LIN {X 0,Y 629.208,Z 740.926,A -85,B 0,C 180,E1 29271.292,E2 29271.292} C_VEL
LIN {X 0,Y 628.174,Z 758.568,A -85,B 0,C 180,E1 29269.915,E2 29269.915} C_VEL
LIN {X 0,Y 627.247,Z 774.118,A -85,B 0,C 180,E1 29268.495,E2 29268.495} C_VEL
LIN {X 0,Y 626.389,Z 788.139,A -85,B 0,C 180,E1 29266.985,E2 29266.985} C_VEL
LIN {X 0,Y 625.582,Z 802.216,A -85,B 0,C 180,E1 29265.196,E2 29265.196} C_VEL
LIN {X 0,Y 624.988,Z 813.341,A -85,B 0,C 180,E1 29263.508,E2 29263.508} C_VEL
LIN {X 0,Y 624.565,Z 822.244,A -85,B 0,C 180,E1 29261.919,E2 29261.919} C_VEL
LIN {X 0,Y 624.211,Z 832.3,A -85,B 0,C 180,E1 29259.776,E2 29259.776} C_VEL
LIN {X 0,Y 624.048,Z 838.961,A -85,B 0,C 180,E1 29258.013,E2 29258.013} C_VEL
LIN {X 0,Y 623.969,Z 843.988,A -85,B 0,C 180,E1 29256.348,E2 29256.348} C_VEL
LIN {X 0,Y 623.918,Z 847.629,A -85,B 0,C 180,E1 29254.78,E2 29254.78} C_VEL
LIN {X 0,Y 623.903,Z 850.253,A -85,B 0,C 180,E1 29253.193,E2 29253.193} C_VEL
LIN {X 0,Y 623.908,Z 851.807,A -85,B 0,C 180,E1 29251.653,E2 29251.653} C_VEL
LIN {X 0,Y 623.919,Z 852.393,A -85,B 0,C 180,E1 29250,E2 29250} C_VEL
LIN {X 0,Y 623.906,Z 851.865,A -85,B 0,C 180,E1 29248.347,E2 29248.347} C_VEL
LIN {X 0,Y 623.901,Z 850.34,A -85,B 0,C 180,E1 29246.785,E2 29246.785} C_VEL
LIN {X 0,Y 623.92,Z 847.804,A -85,B 0,C 180,E1 29245.22,E2 29245.22} C_VEL
LIN {X 0,Y 623.969,Z 844.223,A -85,B 0,C 180,E1 29243.652,E2 29243.652} C_VEL
LIN {X 0,Y 624.029,Z 839.56,A -85,B 0,C 180,E1 29242.08,E2 29242.08} C_VEL
LIN {X 0,Y 624.164,Z 833.767,A -85,B 0,C 180,E1 29240.503,E2 29240.503} C_VEL
LIN {X 0,Y 624.432,Z 825.538,A -85,B 0,C 180,E1 29238.641,E2 29238.641} C_VEL
LIN {X 0,Y 624.9,Z 815.025,A -85,B 0,C 180,E1 29236.679,E2 29236.679} C_VEL
LIN {X 0,Y 625.468,Z 804.166,A -85,B 0,C 180,E1 29234.991,E2 29234.991} C_VEL
LIN {X 0,Y 626.179,Z 791.739,A -85,B 0,C 180,E1 29233.354,E2 29233.354} C_VEL
LIN {X 0,Y 627.018,Z 777.74,A -85,B 0,C 180,E1 29231.787,E2 29231.787} C_VEL
LIN {X 0,Y 627.946,Z 762.367,A -85,B 0,C 180,E1 29230.32,E2 29230.32} C_VEL
LIN {X 0,Y 628.974,Z 745.456,A -85,B 0,C 180,E1 29228.944,E2 29228.944} C_VEL
LIN {X 0,Y 629.98,Z 727.417,A -85,B 0,C 180,E1 29227.708,E2 29227.708} C_VEL
LIN {X 0,Y 630.985,Z 708.54,A -85,B 0,C 180,E1 29226.612,E2 29226.612} C_VEL
LIN {X 0,Y 631.859,Z 689.995,A -85,B 0,C 180,E1 29225.705,E2 29225.705} C_VEL
LIN {X 0,Y 632.742,Z 669.051,A -85,B 0,C 180,E1 29224.87,E2 29224.87} C_VEL
LIN {X 0,Y 633.413,Z 648.623,A -85,B 0,C 180,E1 29224.226,E2 29224.226} C_VEL
LIN {X 0,Y 634.025,Z 626.542,A -85,B 0,C 180,E1 29223.692,E2 29223.692} C_VEL
LIN {X 0,Y 634.453,Z 605.1,A -85,B 0,C 180,E1 29223.321,E2 29223.321} C_VEL
LIN {X 0,Y 638.365,Z 407.202,A -85,B 0,C 180,E1 29220.608,E2 29220.608} C_VEL
LIN {X 0,Y 639.37,Z 326.363,A -85,B 0,C 180,E1 29219.579,E2 29219.579} C_VEL
LIN {X 0,Y 639.015,Z 324.152,A -85,B 0,C 180,E1 29219.511,E2 29219.511} C_VEL
LIN {X 0,Y 639.079,Z 296.354,A -85,B 0,C 180,E1 29217.65,E2 29217.65} C_VEL
LIN {X 0,Y 640.388,Z 256.622,A -85,B 0,C 180,E1 29214.747,E2 29214.747} C_VEL
LIN {X 0,Y 640.643,Z 246.721,A -85,B 0,C 180,E1 29214.024,E2 29214.024} C_VEL
LIN {X 0,Y 633.821,Z 228.869,A -85,B 0,C 180,E1 29212.219,E2 29212.219} C_VEL
LIN {X 0,Y 627.274,Z 213.434,A -85,B 0,C 180,E1 29210.706,E2 29210.706} C_VEL
LIN {X 0,Y 624.952,Z 207.388,A -85,B 0,C 180,E1 29210.129,E2 29210.129} C_VEL
LIN {X 0,Y 624.924,Z 207.385,A -85,B 0,C 180,E1 29206.988,E2 29206.988} C_VEL
LIN {X 0,Y 624.946,Z 207.377,A -85,B 0,C 180,E1 29203.851,E2 29203.851} C_VEL
LIN {X 0,Y 624.928,Z 207.382,A -85,B 0,C 180,E1 29200.754,E2 29200.754} C_VEL
LIN {X 0,Y 624.947,Z 207.376,A -85,B 0,C 180,E1 29197.629,E2 29197.629} C_VEL
LIN {X 0,Y 624.94,Z 207.389,A -85,B 0,C 180,E1 29194.499,E2 29194.499} C_VEL
LIN {X 0,Y 624.947,Z 207.379,A -85,B 0,C 180,E1 29191.224,E2 29191.224} C_VEL
LIN {X 0,Y 624.945,Z 207.373,A -85,B 0,C 180,E1 29188.06,E2 29188.06} C_VEL
LIN {X 0,Y 624.937,Z 207.381,A -85,B 0,C 180,E1 29184.88,E2 29184.88} C_VEL
LIN {X 0,Y 624.937,Z 207.383,A -85,B 0,C 180,E1 29181.79,E2 29181.79} C_VEL
LIN {X 0,Y 624.937,Z 207.371,A -85,B 0,C 180,E1 29178.663,E2 29178.663} C_VEL
LIN {X 0,Y 624.934,Z 207.381,A -85,B 0,C 180,E1 29175.593,E2 29175.593} C_VEL
LIN {X 0,Y 624.941,Z 207.366,A -85,B 0,C 180,E1 29172.474,E2 29172.474} C_VEL
LIN {X 0,Y 624.942,Z 207.38,A -85,B 0,C 180,E1 29169.3,E2 29169.3} C_VEL
LIN {X 0,Y 624.943,Z 207.365,A -85,B 0,C 180,E1 29166.062,E2 29166.062} C_VEL
LIN {X 0,Y 624.947,Z 207.38,A -85,B 0,C 180,E1 29162.843,E2 29162.843} C_VEL
LIN {X 0,Y 624.923,Z 207.363,A -85,B 0,C 180,E1 29159.725,E2 29159.725} C_VEL
LIN {X 0,Y 624.946,Z 207.381,A -85,B 0,C 180,E1 29156.606,E2 29156.606} C_VEL
LIN {X 0,Y 624.919,Z 207.364,A -85,B 0,C 180,E1 29153.477,E2 29153.477} C_VEL
LIN {X 0,Y 624.949,Z 207.381,A -85,B 0,C 180,E1 29150.329,E2 29150.329} C_VEL
LIN {X 0,Y 624.924,Z 207.382,A -85,B 0,C 180,E1 29147.244,E2 29147.244} C_VEL
LIN {X 0,Y 624.942,Z 207.385,A -85,B 0,C 180,E1 29144.026,E2 29144.026} C_VEL
LIN {X 0,Y 624.946,Z 207.377,A -85,B 0,C 180,E1 29140.853,E2 29140.853} C_VEL
LIN {X 0,Y 624.916,Z 207.388,A -85,B 0,C 180,E1 29137.642,E2 29137.642} C_VEL
LIN {X 0,Y 624.953,Z 207.381,A -85,B 0,C 180,E1 29134.609,E2 29134.609} C_VEL
LIN {X 0,Y 624.91,Z 207.385,A -85,B 0,C 180,E1 29131.454,E2 29131.454} C_VEL
LIN {X 0,Y 624.957,Z 207.381,A -85,B 0,C 180,E1 29128.454,E2 29128.454} C_VEL
LIN {X 0,Y 624.906,Z 207.388,A -85,B 0,C 180,E1 29125.329,E2 29125.329} C_VEL
LIN {X 0,Y 624.957,Z 207.38,A -85,B 0,C 180,E1 29122.209,E2 29122.209} C_VEL
LIN {X 0,Y 624.903,Z 207.389,A -85,B 0,C 180,E1 29119.186,E2 29119.186} C_VEL
LIN {X 0,Y 624.95,Z 207.462,A -85,B 0,C 180,E1 29116.613,E2 29116.613} C_VEL
LIN {X 0,Y 626.289,Z 210.904,A -85,B 0,C 180,E1 29116.267,E2 29116.267} C_VEL
LIN {X 0,Y 627.344,Z 212.887,A -85,B 0,C 180,E1 29116.043,E2 29116.043} C_VEL
LIN {X 0,Y 638.156,Z 234.423,A -85,B 0,C 180,E1 29113.754,E2 29113.754} C_VEL
LIN {X 0,Y 647.363,Z 253.935,A -85,B 0,C 180,E1 29111.855,E2 29111.855} C_VEL
LIN {X 0,Y 644.416,Z 304.648,A -85,B 0,C 180,E1 29109.218,E2 29109.218} C_VEL
LIN {X 0,Y 646.898,Z 323.157,A -85,B 0,C 180,E1 29108.795,E2 29108.795} C_VEL
LIN {X 0,Y 644.169,Z 514.087,A -85,B 0,C 180,E1 29106.373,E2 29106.373} C_VEL
LIN {X 0,Y 641.865,Z 692.934,A -85,B 0,C 180,E1 29104.147,E2 29104.147} C_VEL
LIN {X 0,Y 641.079,Z 718.1,A -85,B 0,C 180,E1 29103.674,E2 29103.674} C_VEL
LIN {X 0,Y 640.186,Z 739.868,A -85,B 0,C 180,E1 29103.131,E2 29103.131} C_VEL
LIN {X 0,Y 638.916,Z 765.321,A -85,B 0,C 180,E1 29102.318,E2 29102.318} C_VEL
LIN {X 0,Y 637.689,Z 787.238,A -85,B 0,C 180,E1 29101.461,E2 29101.461} C_VEL
LIN {X 0,Y 636.241,Z 810.546,A -85,B 0,C 180,E1 29100.369,E2 29100.369} C_VEL
LIN {X 0,Y 634.874,Z 830.591,A -85,B 0,C 180,E1 29099.276,E2 29099.276} C_VEL
LIN {X 0,Y 633.292,Z 852.909,A -85,B 0,C 180,E1 29097.862,E2 29097.862} C_VEL
LIN {X 0,Y 632.055,Z 867.818,A -85,B 0,C 180,E1 29096.748,E2 29096.748} C_VEL
LIN {X 0,Y 630.517,Z 886.159,A -85,B 0,C 180,E1 29095.202,E2 29095.202} C_VEL
LIN {X 0,Y 629.035,Z 903.822,A -85,B 0,C 180,E1 29093.482,E2 29093.482} C_VEL
LIN {X 0,Y 627.829,Z 919.315,A -85,B 0,C 180,E1 29091.782,E2 29091.782} C_VEL
LIN {X 0,Y 626.714,Z 934.515,A -85,B 0,C 180,E1 29089.867,E2 29089.867} C_VEL
LIN {X 0,Y 625.867,Z 947.149,A -85,B 0,C 180,E1 29088.055,E2 29088.055} C_VEL
LIN {X 0,Y 625.118,Z 960.283,A -85,B 0,C 180,E1 29085.874,E2 29085.874} C_VEL
LIN {X 0,Y 624.657,Z 970.018,A -85,B 0,C 180,E1 29083.987,E2 29083.987} C_VEL
LIN {X 0,Y 624.293,Z 979.836,A -85,B 0,C 180,E1 29081.736,E2 29081.736} C_VEL
LIN {X 0,Y 624.094,Z 986.816,A -85,B 0,C 180,E1 29079.778,E2 29079.778} C_VEL
LIN {X 0,Y 623.952,Z 993.243,A -85,B 0,C 180,E1 29077.551,E2 29077.551} C_VEL
LIN {X 0,Y 623.905,Z 997.655,A -85,B 0,C 180,E1 29075.426,E2 29075.426} C_VEL
LIN {X 0,Y 623.91,Z 1000.464,A -85,B 0,C 180,E1 29073.491,E2 29073.491} C_VEL
LIN {X 0,Y 623.909,Z 1002.214,A -85,B 0,C 180,E1 29071.194,E2 29071.194} C_VEL
LIN {X 0,Y 623.885,Z 1002.327,A -85,B 0,C 180,E1 29069.265,E2 29069.265} C_VEL
LIN {X 0,Y 623.889,Z 1001.292,A -85,B 0,C 180,E1 29067.336,E2 29067.336} C_VEL
LIN {X 0,Y 623.901,Z 998.451,A -85,B 0,C 180,E1 29065.035,E2 29065.035} C_VEL
LIN {X 0,Y 623.959,Z 994.689,A -85,B 0,C 180,E1 29063.097,E2 29063.097} C_VEL
LIN {X 0,Y 624.042,Z 988.934,A -85,B 0,C 180,E1 29060.873,E2 29060.873} C_VEL
LIN {X 0,Y 624.217,Z 981.602,A -85,B 0,C 180,E1 29058.73,E2 29058.73} C_VEL
LIN {X 0,Y 624.519,Z 973.532,A -85,B 0,C 180,E1 29056.765,E2 29056.765} C_VEL
LIN {X 0,Y 624.996,Z 962.86,A -85,B 0,C 180,E1 29054.599,E2 29054.599} C_VEL
LIN {X 0,Y 625.602,Z 951.969,A -85,B 0,C 180,E1 29052.706,E2 29052.706} C_VEL
LIN {X 0,Y 626.517,Z 937.317,A -85,B 0,C 180,E1 29050.515,E2 29050.515} C_VEL
LIN {X 0,Y 627.462,Z 924.012,A -85,B 0,C 180,E1 29048.785,E2 29048.785} C_VEL
LIN {X 0,Y 628.838,Z 906.301,A -85,B 0,C 180,E1 29046.775,E2 29046.775} C_VEL
LIN {X 0,Y 630.114,Z 890.795,A -85,B 0,C 180,E1 29045.233,E2 29045.233} C_VEL
LIN {X 0,Y 631.805,Z 870.854,A -85,B 0,C 180,E1 29043.494,E2 29043.494} C_VEL
LIN {X 0,Y 633.107,Z 855.309,A -85,B 0,C 180,E1 29042.307,E2 29042.307} C_VEL
LIN {X 0,Y 634.055,Z 841.543,A -85,B 0,C 180,E1 29041.405,E2 29041.405} C_VEL
LIN {X 0,Y 635.449,Z 820.222,A -85,B 0,C 180,E1 29040.183,E2 29040.183} C_VEL
LIN {X 0,Y 636.697,Z 797.901,A -85,B 0,C 180,E1 29039.101,E2 29039.101} C_VEL
LIN {X 0,Y 637.906,Z 775.285,A -85,B 0,C 180,E1 29038.165,E2 29038.165} C_VEL
LIN {X 0,Y 638.944,Z 751.93,A -85,B 0,C 180,E1 29037.377,E2 29037.377} C_VEL
LIN {X 0,Y 639.847,Z 727.921,A -85,B 0,C 180,E1 29036.72,E2 29036.72} C_VEL
LIN {X 0,Y 640.534,Z 703.096,A -85,B 0,C 180,E1 29036.219,E2 29036.219} C_VEL
LIN {X 0,Y 640.998,Z 677.434,A -85,B 0,C 180,E1 29035.856,E2 29035.856} C_VEL
LIN {X 0,Y 642.199,Z 471.258,A -85,B 0,C 180,E1 29033.497,E2 29033.497} C_VEL
LIN {X 0,Y 643.617,Z 320.826,A -85,B 0,C 180,E1 29031.652,E2 29031.652} C_VEL
LIN {X 0,Y 642.214,Z 312.028,A -85,B 0,C 180,E1 29031.452,E2 29031.452} C_VEL
LIN {X 0,Y 644.812,Z 281.295,A -85,B 0,C 180,E1 29029.712,E2 29029.712} C_VEL
LIN {X 0,Y 648.358,Z 254.707,A -85,B 0,C 180,E1 29028.05,E2 29028.05} C_VEL
LIN {X 0,Y 645.178,Z 246.171,A -85,B 0,C 180,E1 29026.883,E2 29026.883} C_VEL
LIN {X 0,Y 642.634,Z 240.116,A -85,B 0,C 180,E1 29025.809,E2 29025.809} C_VEL
LIN {X 0,Y 641.16,Z 236.75,A -85,B 0,C 180,E1 29025.053,E2 29025.053} C_VEL
LIN {X 0,Y 639.826,Z 233.597,A -85,B 0,C 180,E1 29024.168,E2 29024.168} C_VEL
LIN {X 0,Y 638.452,Z 230.647,A -85,B 0,C 180,E1 29022.698,E2 29022.698} C_VEL
LIN {X 0,Y 638.405,Z 229.859,A -85,B 0,C 180,E1 29021.732,E2 29021.732} C_VEL
LIN {X 0,Y 638.414,Z 231.106,A -85,B 0,C 180,E1 29020.658,E2 29020.658} C_VEL
LIN {X 0,Y 639.781,Z 233.899,A -85,B 0,C 180,E1 29019.32,E2 29019.32} C_VEL
LIN {X 0,Y 641.35,Z 238.172,A -85,B 0,C 180,E1 29018.209,E2 29018.209} C_VEL
LIN {X 0,Y 643.354,Z 243.746,A -85,B 0,C 180,E1 29017.127,E2 29017.127} C_VEL
LIN {X 0,Y 645.653,Z 251.249,A -85,B 0,C 180,E1 29016.001,E2 29016.001} C_VEL
LIN {X 0,Y 641.269,Z 281.594,A -85,B 0,C 180,E1 29013.717,E2 29013.717} C_VEL
LIN {X 0,Y 637.312,Z 322.129,A -85,B 0,C 180,E1 29010.885,E2 29010.885} C_VEL
LIN {X 0,Y 634.413,Z 366.282,A -85,B 0,C 180,E1 29007.962,E2 29007.962} C_VEL
LIN {X 0,Y 631.971,Z 416.413,A -85,B 0,C 180,E1 29004.789,E2 29004.789} C_VEL
LIN {X 0,Y 631.044,Z 441.253,A -85,B 0,C 180,E1 29003.28,E2 29003.28} C_VEL
LIN {X 0,Y 635.394,Z 479.453,A -85,B 0,C 180,E1 29002.276,E2 29002.276} C_VEL
LIN {X 0,Y 635.961,Z 488.203,A -85,B 0,C 180,E1 29002.081,E2 29002.081} C_VEL
LIN {X 0,Y 632.244,Z 601.48,A -85,B 0,C 180,E1 29000.279,E2 29000.279} C_VEL
LIN {X 0,Y 630.407,Z 684.522,A -85,B 0,C 180,E1 28999.018,E2 28999.018} C_VEL
LIN {X 0,Y 629.845,Z 705.803,A -85,B 0,C 180,E1 28998.518,E2 28998.518} C_VEL
LIN {X 0,Y 629.291,Z 724.826,A -85,B 0,C 180,E1 28997.906,E2 28997.906} C_VEL
LIN {X 0,Y 628.646,Z 743.951,A -85,B 0,C 180,E1 28997.113,E2 28997.113} C_VEL
LIN {X 0,Y 628.049,Z 760.98,A -85,B 0,C 180,E1 28996.23,E2 28996.23} C_VEL
LIN {X 0,Y 627.432,Z 777.32,A -85,B 0,C 180,E1 28995.198,E2 28995.198} C_VEL
LIN {X 0,Y 626.858,Z 791.603,A -85,B 0,C 180,E1 28994.114,E2 28994.114} C_VEL
LIN {X 0,Y 626.317,Z 804.831,A -85,B 0,C 180,E1 28992.915,E2 28992.915} C_VEL
LIN {X 0,Y 625.835,Z 816.839,A -85,B 0,C 180,E1 28991.614,E2 28991.614} C_VEL
LIN {X 0,Y 625.39,Z 828.124,A -85,B 0,C 180,E1 28990.129,E2 28990.129} C_VEL
LIN {X 0,Y 625.031,Z 837.79,A -85,B 0,C 180,E1 28988.556,E2 28988.556} C_VEL
LIN {X 0,Y 624.78,Z 845.408,A -85,B 0,C 180,E1 28986.986,E2 28986.986} C_VEL
LIN {X 0,Y 624.611,Z 851.521,A -85,B 0,C 180,E1 28985.327,E2 28985.327} C_VEL
LIN {X 0,Y 624.48,Z 855.819,A -85,B 0,C 180,E1 28983.672,E2 28983.672} C_VEL
LIN {X 0,Y 624.401,Z 858.528,A -85,B 0,C 180,E1 28981.927,E2 28981.927} C_VEL
LIN {X 0,Y 624.361,Z 859.436,A -85,B 0,C 180,E1 28980.184,E2 28980.184} C_VEL
LIN {X 0,Y 624.335,Z 858.578,A -85,B 0,C 180,E1 28978.44,E2 28978.44} C_VEL
LIN {X 0,Y 624.355,Z 855.951,A -85,B 0,C 180,E1 28976.695,E2 28976.695} C_VEL
LIN {X 0,Y 624.419,Z 851.496,A -85,B 0,C 180,E1 28974.947,E2 28974.947} C_VEL
LIN {X 0,Y 624.534,Z 845.462,A -85,B 0,C 180,E1 28973.288,E2 28973.288} C_VEL
LIN {X 0,Y 624.739,Z 837.497,A -85,B 0,C 180,E1 28971.625,E2 28971.625} C_VEL
LIN {X 0,Y 625.04,Z 827.956,A -85,B 0,C 180,E1 28970.051,E2 28970.051} C_VEL
LIN {X 0,Y 625.447,Z 816.489,A -85,B 0,C 180,E1 28968.52,E2 28968.52} C_VEL
LIN {X 0,Y 625.919,Z 804.267,A -85,B 0,C 180,E1 28967.171,E2 28967.171} C_VEL
LIN {X 0,Y 626.493,Z 790.059,A -85,B 0,C 180,E1 28965.866,E2 28965.866} C_VEL
LIN {X 0,Y 627.113,Z 775.015,A -85,B 0,C 180,E1 28964.717,E2 28964.717} C_VEL
LIN {X 0,Y 627.76,Z 758.503,A -85,B 0,C 180,E1 28963.672,E2 28963.672} C_VEL
LIN {X 0,Y 628.401,Z 741.33,A -85,B 0,C 180,E1 28962.785,E2 28962.785} C_VEL
LIN {X 0,Y 629.033,Z 723.273,A -85,B 0,C 180,E1 28962.039,E2 28962.039} C_VEL
LIN {X 0,Y 629.604,Z 703.456,A -85,B 0,C 180,E1 28961.412,E2 28961.412} C_VEL
LIN {X 0,Y 630.065,Z 683.762,A -85,B 0,C 180,E1 28960.969,E2 28960.969} C_VEL
LIN {X 0,Y 630.481,Z 653.884,A -85,B 0,C 180,E1 28960.552,E2 28960.552} C_VEL
LIN {X 0,Y 632.813,Z 483.695,A -85,B 0,C 180,E1 28958.323,E2 28958.323} C_VEL
LIN {X 0,Y 630.114,Z 460.538,A -85,B 0,C 180,E1 28957.865,E2 28957.865} C_VEL
LIN {X 0,Y 631.884,Z 406.271,A -85,B 0,C 180,E1 28954.607,E2 28954.607} C_VEL
LIN {X 0,Y 632.169,Z 397.972,A -85,B 0,C 180,E1 28954.106,E2 28954.106} C_VEL
LIN {X 0,Y 631.485,Z 391.743,A -85,B 0,C 180,E1 28953.69,E2 28953.69} C_VEL
LIN {X 0,Y 626.328,Z 376.015,A -85,B 0,C 180,E1 28952.474,E2 28952.474} C_VEL
LIN {X 0,Y 625.851,Z 370.657,A -85,B 0,C 180,E1 28952.113,E2 28952.113} C_VEL
LIN {X 0,Y 627.881,Z 321.996,A -85,B 0,C 180,E1 28949.098,E2 28949.098} C_VEL
LIN {X 0,Y 630.347,Z 269.288,A -85,B 0,C 180,E1 28945.777,E2 28945.777} C_VEL
LIN {X 0,Y 631.298,Z 245.645,A -85,B 0,C 180,E1 28944.258,E2 28944.258} C_VEL
LIN {X 0,Y 620.877,Z 218.382,A -85,B 0,C 180,E1 28941.729,E2 28941.729} C_VEL
LIN {X 0,Y 616.989,Z 208.38,A -85,B 0,C 180,E1 28940.754,E2 28940.754} C_VEL
LIN {X 0,Y 616.96,Z 208.381,A -85,B 0,C 180,E1 28937.649,E2 28937.649} C_VEL
LIN {X 0,Y 617.013,Z 208.37,A -85,B 0,C 180,E1 28934.517,E2 28934.517} C_VEL
LIN {X 0,Y 616.977,Z 208.375,A -85,B 0,C 180,E1 28931.379,E2 28931.379} C_VEL
LIN {X 0,Y 617.033,Z 208.453,A -85,B 0,C 180,E1 28930.27,E2 28930.27} C_VEL
LIN {X 0,Y 618.333,Z 211.922,A -85,B 0,C 180,E1 28929.96,E2 28929.96} C_VEL
LIN {X 0,Y 625.978,Z 229.789,A -85,B 0,C 180,E1 28928.197,E2 28928.197} C_VEL
LIN {X 0,Y 633.173,Z 248.32,A -85,B 0,C 180,E1 28926.313,E2 28926.313} C_VEL
LIN {X 0,Y 633.844,Z 251.207,A -85,B 0,C 180,E1 28926.044,E2 28926.044} C_VEL
LIN {X 0,Y 632.416,Z 295.085,A -85,B 0,C 180,E1 28922.841,E2 28922.841} C_VEL
LIN {X 0,Y 632.309,Z 325.01,A -85,B 0,C 180,E1 28920.833,E2 28920.833} C_VEL
LIN {X 0,Y 632.515,Z 327.844,A -85,B 0,C 180,E1 28920.687,E2 28920.687} C_VEL
LIN {X 0,Y 631.027,Z 428.42,A -85,B 0,C 180,E1 28919.385,E2 28919.385} C_VEL
LIN {X 0,Y 627.72,Z 572.114,A -85,B 0,C 180,E1 28917.337,E2 28917.337} C_VEL
LIN {X 0,Y 626.665,Z 621.823,A -85,B 0,C 180,E1 28916.577,E2 28916.577} C_VEL
LIN {X 0,Y 626.054,Z 644.64,A -85,B 0,C 180,E1 28916.054,E2 28916.054} C_VEL
LIN {X 0,Y 625.271,Z 666.522,A -85,B 0,C 180,E1 28915.376,E2 28915.376} C_VEL
LIN {X 0,Y 624.38,Z 687.651,A -85,B 0,C 180,E1 28914.549,E2 28914.549} C_VEL
LIN {X 0,Y 623.372,Z 708.562,A -85,B 0,C 180,E1 28913.541,E2 28913.541} C_VEL
LIN {X 0,Y 622.343,Z 727.705,A -85,B 0,C 180,E1 28912.432,E2 28912.432} C_VEL
LIN {X 0,Y 621.33,Z 745.237,A -85,B 0,C 180,E1 28911.229,E2 28911.229} C_VEL
LIN {X 0,Y 620.289,Z 761.787,A -85,B 0,C 180,E1 28909.885,E2 28909.885} C_VEL
LIN {X 0,Y 619.288,Z 777.907,A -85,B 0,C 180,E1 28908.351,E2 28908.351} C_VEL
LIN {X 0,Y 618.441,Z 791.683,A -85,B 0,C 180,E1 28906.822,E2 28906.822} C_VEL
LIN {X 0,Y 617.705,Z 804.058,A -85,B 0,C 180,E1 28905.203,E2 28905.203} C_VEL
LIN {X 0,Y 617.096,Z 815.114,A -85,B 0,C 180,E1 28903.493,E2 28903.493} C_VEL
LIN {X 0,Y 616.602,Z 825.387,A -85,B 0,C 180,E1 28901.6,E2 28901.6} C_VEL
LIN {X 0,Y 616.252,Z 834.032,A -85,B 0,C 180,E1 28899.621,E2 28899.621} C_VEL
LIN {X 0,Y 616.054,Z 840.215,A -85,B 0,C 180,E1 28897.836,E2 28897.836} C_VEL
LIN {X 0,Y 615.975,Z 844.61,A -85,B 0,C 180,E1 28896.244,E2 28896.244} C_VEL
LIN {X 0,Y 615.929,Z 848.876,A -85,B 0,C 180,E1 28894.189,E2 28894.189} C_VEL
LIN {X 0,Y 615.916,Z 851.625,A -85,B 0,C 180,E1 28891.954,E2 28891.954} C_VEL
LIN {X 0,Y 615.906,Z 852.387,A -85,B 0,C 180,E1 28890.186,E2 28890.186} C_VEL
LIN {X 0,Y 615.899,Z 851.978,A -85,B 0,C 180,E1 28888.512,E2 28888.512} C_VEL
LIN {X 0,Y 615.902,Z 850.572,A -85,B 0,C 180,E1 28886.929,E2 28886.929} C_VEL
LIN {X 0,Y 615.924,Z 848.154,A -85,B 0,C 180,E1 28885.344,E2 28885.344} C_VEL
LIN {X 0,Y 615.977,Z 844.374,A -85,B 0,C 180,E1 28883.569,E2 28883.569} C_VEL
LIN {X 0,Y 616.076,Z 839.628,A -85,B 0,C 180,E1 28881.883,E2 28881.883} C_VEL
LIN {X 0,Y 616.312,Z 832.537,A -85,B 0,C 180,E1 28879.909,E2 28879.909} C_VEL
LIN {X 0,Y 616.686,Z 823.437,A -85,B 0,C 180,E1 28877.927,E2 28877.927} C_VEL
LIN {X 0,Y 617.192,Z 813.408,A -85,B 0,C 180,E1 28876.127,E2 28876.127} C_VEL
LIN {X 0,Y 617.822,Z 801.948,A -85,B 0,C 180,E1 28874.416,E2 28874.416} C_VEL
LIN {X 0,Y 618.63,Z 788.345,A -85,B 0,C 180,E1 28872.699,E2 28872.699} C_VEL
LIN {X 0,Y 619.532,Z 774.136,A -85,B 0,C 180,E1 28871.168,E2 28871.168} C_VEL
LIN {X 0,Y 620.513,Z 758.369,A -85,B 0,C 180,E1 28869.73,E2 28869.73} C_VEL
LIN {X 0,Y 621.556,Z 741.112,A -85,B 0,C 180,E1 28868.384,E2 28868.384} C_VEL
LIN {X 0,Y 622.603,Z 723.132,A -85,B 0,C 180,E1 28867.197,E2 28867.197} C_VEL
LIN {X 0,Y 623.623,Z 703.837,A -85,B 0,C 180,E1 28866.118,E2 28866.118} C_VEL
LIN {X 0,Y 624.567,Z 683.722,A -85,B 0,C 180,E1 28865.194,E2 28865.194} C_VEL
LIN {X 0,Y 625.368,Z 663.257,A -85,B 0,C 180,E1 28864.425,E2 28864.425} C_VEL
LIN {X 0,Y 626.144,Z 641.208,A -85,B 0,C 180,E1 28863.771,E2 28863.771} C_VEL
LIN {X 0,Y 626.707,Z 619.44,A -85,B 0,C 180,E1 28863.288,E2 28863.288} C_VEL
LIN {X 0,Y 630.374,Z 458.135,A -85,B 0,C 180,E1 28860.933,E2 28860.933} C_VEL
LIN {X 0,Y 632.296,Z 356.258,A -85,B 0,C 180,E1 28859.587,E2 28859.587} C_VEL
LIN {X 0,Y 632.526,Z 327.84,A -85,B 0,C 180,E1 28859.223,E2 28859.223} C_VEL
LIN {X 0,Y 632.323,Z 325.004,A -85,B 0,C 180,E1 28859.075,E2 28859.075} C_VEL
LIN {X 0,Y 632.406,Z 297.282,A -85,B 0,C 180,E1 28857.218,E2 28857.218} C_VEL
LIN {X 0,Y 633.772,Z 254.797,A -85,B 0,C 180,E1 28854.119,E2 28854.119} C_VEL
LIN {X 0,Y 633.892,Z 250.34,A -85,B 0,C 180,E1 28853.788,E2 28853.788} C_VEL
LIN {X 0,Y 625.98,Z 229.699,A -85,B 0,C 180,E1 28851.701,E2 28851.701} C_VEL
LIN {X 0,Y 618.297,Z 211.831,A -85,B 0,C 180,E1 28849.937,E2 28849.937} C_VEL
LIN {X 0,Y 617.017,Z 208.37,A -85,B 0,C 180,E1 28849.593,E2 28849.593} C_VEL
LIN {X 0,Y 617.009,Z 208.367,A -85,B 0,C 180,E1 28846.342,E2 28846.342} C_VEL
LIN {X 0,Y 616.992,Z 208.368,A -85,B 0,C 180,E1 28843.149,E2 28843.149} C_VEL
LIN {X 0,Y 617.007,Z 208.367,A -85,B 0,C 180,E1 28840.043,E2 28840.043} C_VEL
LIN {X 0,Y 616.992,Z 208.364,A -85,B 0,C 180,E1 28836.959,E2 28836.959} C_VEL
LIN {X 0,Y 617.003,Z 208.365,A -85,B 0,C 180,E1 28833.881,E2 28833.881} C_VEL
LIN {X 0,Y 616.995,Z 208.374,A -85,B 0,C 180,E1 28830.696,E2 28830.696} C_VEL
LIN {X 0,Y 617.008,Z 208.365,A -85,B 0,C 180,E1 28827.507,E2 28827.507} C_VEL
LIN {X 0,Y 617.009,Z 208.359,A -85,B 0,C 180,E1 28824.307,E2 28824.307} C_VEL
LIN {X 0,Y 617.008,Z 208.367,A -85,B 0,C 180,E1 28821.023,E2 28821.023} C_VEL
LIN {X 0,Y 616.996,Z 208.355,A -85,B 0,C 180,E1 28817.836,E2 28817.836} C_VEL
LIN {X 0,Y 617.001,Z 208.372,A -85,B 0,C 180,E1 28814.652,E2 28814.652} C_VEL
LIN {X 0,Y 616.993,Z 208.359,A -85,B 0,C 180,E1 28811.498,E2 28811.498} C_VEL
LIN {X 0,Y 617.011,Z 208.373,A -85,B 0,C 180,E1 28808.293,E2 28808.293} C_VEL
LIN {X 0,Y 617.008,Z 208.354,A -85,B 0,C 180,E1 28805.02,E2 28805.02} C_VEL
LIN {X 0,Y 616.993,Z 208.37,A -85,B 0,C 180,E1 28801.857,E2 28801.857} C_VEL
LIN {X 0,Y 617.007,Z 208.349,A -85,B 0,C 180,E1 28798.7,E2 28798.7} C_VEL
LIN {X 0,Y 616.985,Z 208.371,A -85,B 0,C 180,E1 28795.538,E2 28795.538} C_VEL
LIN {X 0,Y 617.009,Z 208.349,A -85,B 0,C 180,E1 28792.364,E2 28792.364} C_VEL
LIN {X 0,Y 616.987,Z 208.371,A -85,B 0,C 180,E1 28789.259,E2 28789.259} C_VEL
LIN {X 0,Y 617.006,Z 208.376,A -85,B 0,C 180,E1 28786.027,E2 28786.027} C_VEL
LIN {X 0,Y 617.009,Z 208.37,A -85,B 0,C 180,E1 28782.846,E2 28782.846} C_VEL
LIN {X 0,Y 616.982,Z 208.375,A -85,B 0,C 180,E1 28779.707,E2 28779.707} C_VEL
LIN {X 0,Y 617.018,Z 208.372,A -85,B 0,C 180,E1 28776.607,E2 28776.607} C_VEL
LIN {X 0,Y 616.971,Z 208.37,A -85,B 0,C 180,E1 28773.429,E2 28773.429} C_VEL
LIN {X 0,Y 617.019,Z 208.369,A -85,B 0,C 180,E1 28770.296,E2 28770.296} C_VEL
LIN {X 0,Y 616.969,Z 208.376,A -85,B 0,C 180,E1 28767.228,E2 28767.228} C_VEL
LIN {X 0,Y 617.008,Z 208.37,A -85,B 0,C 180,E1 28764.081,E2 28764.081} C_VEL
LIN {X 0,Y 616.97,Z 208.376,A -85,B 0,C 180,E1 28761.037,E2 28761.037} C_VEL
LIN {X 0,Y 616.984,Z 208.374,A -85,B 0,C 180,E1 28757.784,E2 28757.784} C_VEL
LIN {X 0,Y 616.973,Z 208.473,A -85,B 0,C 180,E1 28757.279,E2 28757.279} C_VEL
LIN {X 0,Y 618.159,Z 211.679,A -85,B 0,C 180,E1 28756.953,E2 28756.953} C_VEL
LIN {X 0,Y 619.445,Z 213.94,A -85,B 0,C 180,E1 28756.684,E2 28756.684} C_VEL
LIN {X 0,Y 630.352,Z 235.7,A -85,B 0,C 180,E1 28754.324,E2 28754.324} C_VEL
LIN {X 0,Y 640.346,Z 256.314,A -85,B 0,C 180,E1 28752.256,E2 28752.256} C_VEL
LIN {X 0,Y 640.785,Z 257.643,A -85,B 0,C 180,E1 28752.143,E2 28752.143} C_VEL
LIN {X 0,Y 637.808,Z 305.28,A -85,B 0,C 180,E1 28749.637,E2 28749.637} C_VEL
LIN {X 0,Y 640.349,Z 324.485,A -85,B 0,C 180,E1 28749.193,E2 28749.193} C_VEL
LIN {X 0,Y 637.351,Z 514.536,A -85,B 0,C 180,E1 28746.745,E2 28746.745} C_VEL
LIN {X 0,Y 634.819,Z 693.056,A -85,B 0,C 180,E1 28744.488,E2 28744.488} C_VEL
LIN {X 0,Y 633.989,Z 718.022,A -85,B 0,C 180,E1 28744.014,E2 28744.014} C_VEL
LIN {X 0,Y 633.043,Z 739.755,A -85,B 0,C 180,E1 28743.465,E2 28743.465} C_VEL
LIN {X 0,Y 631.732,Z 764.586,A -85,B 0,C 180,E1 28742.665,E2 28742.665} C_VEL
LIN {X 0,Y 630.423,Z 786.292,A -85,B 0,C 180,E1 28741.811,E2 28741.811} C_VEL
LIN {X 0,Y 628.88,Z 810.034,A -85,B 0,C 180,E1 28740.689,E2 28740.689} C_VEL
LIN {X 0,Y 627.456,Z 829.744,A -85,B 0,C 180,E1 28739.604,E2 28739.604} C_VEL
LIN {X 0,Y 625.763,Z 852.12,A -85,B 0,C 180,E1 28738.175,E2 28738.175} C_VEL
LIN {X 0,Y 624.347,Z 870.25,A -85,B 0,C 180,E1 28736.848,E2 28736.848} C_VEL
LIN {X 0,Y 622.966,Z 887.246,A -85,B 0,C 180,E1 28735.426,E2 28735.426} C_VEL
LIN {X 0,Y 621.405,Z 904.515,A -85,B 0,C 180,E1 28733.713,E2 28733.713} C_VEL
LIN {X 0,Y 620.037,Z 920.984,A -85,B 0,C 180,E1 28731.871,E2 28731.871} C_VEL
LIN {X 0,Y 618.856,Z 935.914,A -85,B 0,C 180,E1 28729.933,E2 28729.933} C_VEL
LIN {X 0,Y 617.897,Z 949.659,A -85,B 0,C 180,E1 28727.906,E2 28727.906} C_VEL
LIN {X 0,Y 617.171,Z 961.311,A -85,B 0,C 180,E1 28725.89,E2 28725.89} C_VEL
LIN {X 0,Y 616.667,Z 971.394,A -85,B 0,C 180,E1 28723.885,E2 28723.885} C_VEL
LIN {X 0,Y 616.3,Z 980.543,A -85,B 0,C 180,E1 28721.701,E2 28721.701} C_VEL
LIN {X 0,Y 616.105,Z 987.119,A -85,B 0,C 180,E1 28719.811,E2 28719.811} C_VEL
LIN {X 0,Y 615.955,Z 993.45,A -85,B 0,C 180,E1 28717.556,E2 28717.556} C_VEL
LIN {X 0,Y 615.909,Z 997.654,A -85,B 0,C 180,E1 28715.496,E2 28715.496} C_VEL
LIN {X 0,Y 615.912,Z 1000.464,A -85,B 0,C 180,E1 28713.537,E2 28713.537} C_VEL
LIN {X 0,Y 615.909,Z 1002.214,A -85,B 0,C 180,E1 28711.209,E2 28711.209} C_VEL
LIN {X 0,Y 615.887,Z 1002.327,A -85,B 0,C 180,E1 28709.256,E2 28709.256} C_VEL
LIN {X 0,Y 615.888,Z 1001.291,A -85,B 0,C 180,E1 28707.301,E2 28707.301} C_VEL
LIN {X 0,Y 615.901,Z 998.451,A -85,B 0,C 180,E1 28704.971,E2 28704.971} C_VEL
LIN {X 0,Y 615.968,Z 994.689,A -85,B 0,C 180,E1 28703.007,E2 28703.007} C_VEL
LIN {X 0,Y 616.063,Z 988.934,A -85,B 0,C 180,E1 28700.754,E2 28700.754} C_VEL
LIN {X 0,Y 616.25,Z 981.601,A -85,B 0,C 180,E1 28698.583,E2 28698.583} C_VEL
LIN {X 0,Y 616.573,Z 973.534,A -85,B 0,C 180,E1 28696.591,E2 28696.591} C_VEL
LIN {X 0,Y 617.093,Z 962.859,A -85,B 0,C 180,E1 28694.397,E2 28694.397} C_VEL
LIN {X 0,Y 617.754,Z 951.968,A -85,B 0,C 180,E1 28692.479,E2 28692.479} C_VEL
LIN {X 0,Y 618.754,Z 937.315,A -85,B 0,C 180,E1 28690.261,E2 28690.261} C_VEL
LIN {X 0,Y 619.76,Z 924.072,A -85,B 0,C 180,E1 28688.517,E2 28688.517} C_VEL
LIN {X 0,Y 621.184,Z 907.148,A -85,B 0,C 180,E1 28686.564,E2 28686.564} C_VEL
LIN {X 0,Y 622.531,Z 891.808,A -85,B 0,C 180,E1 28685.012,E2 28685.012} C_VEL
LIN {X 0,Y 623.751,Z 877.634,A -85,B 0,C 180,E1 28683.741,E2 28683.741} C_VEL
LIN {X 0,Y 625.28,Z 857.186,A -85,B 0,C 180,E1 28682.216,E2 28682.216} C_VEL
LIN {X 0,Y 626.602,Z 838.163,A -85,B 0,C 180,E1 28680.981,E2 28680.981} C_VEL
LIN {X 0,Y 628.135,Z 814.525,A -85,B 0,C 180,E1 28679.658,E2 28679.658} C_VEL
LIN {X 0,Y 629.406,Z 793.652,A -85,B 0,C 180,E1 28678.664,E2 28678.664} C_VEL
LIN {X 0,Y 630.686,Z 768.887,A -85,B 0,C 180,E1 28677.674,E2 28677.674} C_VEL
LIN {X 0,Y 631.695,Z 746.627,A -85,B 0,C 180,E1 28676.948,E2 28676.948} C_VEL
LIN {X 0,Y 632.655,Z 721.058,A -85,B 0,C 180,E1 28676.293,E2 28676.293} C_VEL
LIN {X 0,Y 633.288,Z 698.869,A -85,B 0,C 180,E1 28675.868,E2 28675.868} C_VEL
LIN {X 0,Y 633.718,Z 665.184,A -85,B 0,C 180,E1 28675.434,E2 28675.434} C_VEL
LIN {X 0,Y 634.955,Z 479.261,A -85,B 0,C 180,E1 28673.275,E2 28673.275} C_VEL
LIN {X 0,Y 636.703,Z 327.978,A -85,B 0,C 180,E1 28671.377,E2 28671.377} C_VEL
LIN {X 0,Y 636.546,Z 320.962,A -85,B 0,C 180,E1 28671.27,E2 28671.27} C_VEL
LIN {X 0,Y 635.484,Z 314.12,A -85,B 0,C 180,E1 28671.112,E2 28671.112} C_VEL
LIN {X 0,Y 638.266,Z 285.583,A -85,B 0,C 180,E1 28669.446,E2 28669.446} C_VEL
LIN {X 0,Y 642.169,Z 259.764,A -85,B 0,C 180,E1 28667.788,E2 28667.788} C_VEL
LIN {X 0,Y 642.228,Z 258.59,A -85,B 0,C 180,E1 28667.692,E2 28667.692} C_VEL
LIN {X 0,Y 639.122,Z 249.943,A -85,B 0,C 180,E1 28666.415,E2 28666.415} C_VEL
LIN {X 0,Y 636.649,Z 243.671,A -85,B 0,C 180,E1 28665.156,E2 28665.156} C_VEL
LIN {X 0,Y 635.084,Z 239.999,A -85,B 0,C 180,E1 28664.099,E2 28664.099} C_VEL
LIN {X 0,Y 633.833,Z 237.204,A -85,B 0,C 180,E1 28662.682,E2 28662.682} C_VEL
LIN {X 0,Y 633.8,Z 236.401,A -85,B 0,C 180,E1 28661.737,E2 28661.737} C_VEL
LIN {X 0,Y 633.762,Z 237.707,A -85,B 0,C 180,E1 28660.635,E2 28660.635} C_VEL
LIN {X 0,Y 634.883,Z 240.241,A -85,B 0,C 180,E1 28659.397,E2 28659.397} C_VEL
LIN {X 0,Y 636.359,Z 244.575,A -85,B 0,C 180,E1 28658.249,E2 28658.249} C_VEL
LIN {X 0,Y 638.32,Z 250.537,A -85,B 0,C 180,E1 28657.091,E2 28657.091} C_VEL
LIN {X 0,Y 639.719,Z 255.46,A -85,B 0,C 180,E1 28656.326,E2 28656.326} C_VEL
LIN {X 0,Y 635.013,Z 284.273,A -85,B 0,C 180,E1 28654.095,E2 28654.095} C_VEL
LIN {X 0,Y 630.81,Z 322.111,A -85,B 0,C 180,E1 28651.38,E2 28651.38} C_VEL
LIN {X 0,Y 627.539,Z 365.868,A -85,B 0,C 180,E1 28648.414,E2 28648.414} C_VEL
LIN {X 0,Y 624.783,Z 415.762,A -85,B 0,C 180,E1 28645.195,E2 28645.195} C_VEL
LIN {X 0,Y 623.838,Z 438.254,A -85,B 0,C 180,E1 28643.806,E2 28643.806} C_VEL
LIN {X 0,Y 627.937,Z 474.401,A -85,B 0,C 180,E1 28642.796,E2 28642.796} C_VEL
LIN {X 0,Y 629.105,Z 489.006,A -85,B 0,C 180,E1 28642.448,E2 28642.448} C_VEL
LIN {X 0,Y 625.251,Z 593.403,A -85,B 0,C 180,E1 28640.721,E2 28640.721} C_VEL
LIN {X 0,Y 622.958,Z 685.281,A -85,B 0,C 180,E1 28639.278,E2 28639.278} C_VEL
LIN {X 0,Y 622.336,Z 706.835,A -85,B 0,C 180,E1 28638.756,E2 28638.756} C_VEL
LIN {X 0,Y 621.709,Z 726.543,A -85,B 0,C 180,E1 28638.102,E2 28638.102} C_VEL
LIN {X 0,Y 621.011,Z 745.815,A -85,B 0,C 180,E1 28637.281,E2 28637.281} C_VEL
LIN {X 0,Y 620.384,Z 762.755,A -85,B 0,C 180,E1 28636.383,E2 28636.383} C_VEL
LIN {X 0,Y 619.731,Z 778.89,A -85,B 0,C 180,E1 28635.343,E2 28635.343} C_VEL
LIN {X 0,Y 619.102,Z 793.493,A -85,B 0,C 180,E1 28634.211,E2 28634.211} C_VEL
LIN {X 0,Y 618.525,Z 806.716,A -85,B 0,C 180,E1 28632.986,E2 28632.986} C_VEL
LIN {X 0,Y 618.015,Z 818.608,A -85,B 0,C 180,E1 28631.668,E2 28631.668} C_VEL
LIN {X 0,Y 617.567,Z 829.154,A -85,B 0,C 180,E1 28630.259,E2 28630.259} C_VEL
LIN {X 0,Y 617.196,Z 838.337,A -85,B 0,C 180,E1 28628.759,E2 28628.759} C_VEL
LIN {X 0,Y 616.912,Z 846.081,A -85,B 0,C 180,E1 28627.169,E2 28627.169} C_VEL
LIN {X 0,Y 616.715,Z 852.453,A -85,B 0,C 180,E1 28625.443,E2 28625.443} C_VEL
LIN {X 0,Y 616.566,Z 856.904,A -85,B 0,C 180,E1 28623.719,E2 28623.719} C_VEL
LIN {X 0,Y 616.479,Z 859.501,A -85,B 0,C 180,E1 28622.045,E2 28622.045} C_VEL
LIN {X 0,Y 616.431,Z 860.478,A -85,B 0,C 180,E1 28620.279,E2 28620.279} C_VEL
LIN {X 0,Y 616.404,Z 859.673,A -85,B 0,C 180,E1 28618.513,E2 28618.513} C_VEL
LIN {X 0,Y 616.42,Z 857.088,A -85,B 0,C 180,E1 28616.745,E2 28616.745} C_VEL
LIN {X 0,Y 616.483,Z 852.666,A -85,B 0,C 180,E1 28614.975,E2 28614.975} C_VEL
LIN {X 0,Y 616.605,Z 846.665,A -85,B 0,C 180,E1 28613.295,E2 28613.295} C_VEL
LIN {X 0,Y 616.819,Z 838.736,A -85,B 0,C 180,E1 28611.611,E2 28611.611} C_VEL
LIN {X 0,Y 617.137,Z 829.244,A -85,B 0,C 180,E1 28610.017,E2 28610.017} C_VEL
LIN {X 0,Y 617.555,Z 818.24,A -85,B 0,C 180,E1 28608.513,E2 28608.513} C_VEL
LIN {X 0,Y 618.065,Z 805.716,A -85,B 0,C 180,E1 28607.1,E2 28607.1} C_VEL
LIN {X 0,Y 618.669,Z 791.613,A -85,B 0,C 180,E1 28605.779,E2 28605.779} C_VEL
LIN {X 0,Y 619.328,Z 776.469,A -85,B 0,C 180,E1 28604.598,E2 28604.598} C_VEL
LIN {X 0,Y 620.028,Z 759.586,A -85,B 0,C 180,E1 28603.511,E2 28603.511} C_VEL
LIN {X 0,Y 620.715,Z 742.199,A -85,B 0,C 180,E1 28602.598,E2 28602.598} C_VEL
LIN {X 0,Y 621.41,Z 723.397,A -85,B 0,C 180,E1 28601.811,E2 28601.811} C_VEL
LIN {X 0,Y 622.019,Z 703.449,A -85,B 0,C 180,E1 28601.173,E2 28601.173} C_VEL
LIN {X 0,Y 622.515,Z 683.599,A -85,B 0,C 180,E1 28600.723,E2 28600.723} C_VEL
LIN {X 0,Y 622.953,Z 653.668,A -85,B 0,C 180,E1 28600.302,E2 28600.302} C_VEL
LIN {X 0,Y 625.477,Z 484.522,A -85,B 0,C 180,E1 28598.036,E2 28598.036} C_VEL
LIN {X 0,Y 622.598,Z 459.59,A -85,B 0,C 180,E1 28597.528,E2 28597.528} C_VEL
LIN {X 0,Y 624.439,Z 406.912,A -85,B 0,C 180,E1 28594.333,E2 28594.333} C_VEL
LIN {X 0,Y 625.851,Z 370.657,A -85,B 0,C 180,E1 28592.113,E2 28592.113} C_VEL
LIN {X 0,Y 625.208,Z 364.456,A -85,B 0,C 180,E1 28591.689,E2 28591.689} C_VEL
LIN {X 0,Y 620.194,Z 348.83,A -85,B 0,C 180,E1 28590.444,E2 28590.444} C_VEL
LIN {X 0,Y 619.749,Z 343.494,A -85,B 0,C 180,E1 28590.076,E2 28590.076} C_VEL
LIN {X 0,Y 622.209,Z 291.194,A -85,B 0,C 180,E1 28586.771,E2 28586.771} C_VEL
LIN {X 0,Y 624.317,Z 248.989,A -85,B 0,C 180,E1 28584.057,E2 28584.057} C_VEL
LIN {X 0,Y 614.323,Z 222.767,A -85,B 0,C 180,E1 28581.601,E2 28581.601} C_VEL
LIN {X 0,Y 609.048,Z 209.364,A -85,B 0,C 180,E1 28580.264,E2 28580.264} C_VEL
LIN {X 0,Y 609.051,Z 209.365,A -85,B 0,C 180,E1 28577.182,E2 28577.182} C_VEL
LIN {X 0,Y 609.064,Z 209.364,A -85,B 0,C 180,E1 28573.982,E2 28573.982} C_VEL
LIN {X 0,Y 609.038,Z 209.363,A -85,B 0,C 180,E1 28570.924,E2 28570.924} C_VEL
LIN {X 0,Y 609.065,Z 209.524,A -85,B 0,C 180,E1 28570.815,E2 28570.815} C_VEL
LIN {X 0,Y 610.316,Z 212.754,A -85,B 0,C 180,E1 28570.52,E2 28570.52} C_VEL
LIN {X 0,Y 618.228,Z 230.9,A -85,B 0,C 180,E1 28568.705,E2 28568.705} C_VEL
LIN {X 0,Y 625.536,Z 249.642,A -85,B 0,C 180,E1 28566.791,E2 28566.791} C_VEL
LIN {X 0,Y 627.086,Z 254.149,A -85,B 0,C 180,E1 28566.33,E2 28566.33} C_VEL
LIN {X 0,Y 625.713,Z 298.975,A -85,B 0,C 180,E1 28563.074,E2 28563.074} C_VEL
LIN {X 0,Y 625.687,Z 327.356,A -85,B 0,C 180,E1 28561.183,E2 28561.183} C_VEL
LIN {X 0,Y 625.859,Z 330.298,A -85,B 0,C 180,E1 28561.029,E2 28561.029} C_VEL
LIN {X 0,Y 623.942,Z 436.328,A -85,B 0,C 180,E1 28559.647,E2 28559.647} C_VEL
LIN {X 0,Y 620.804,Z 560.124,A -85,B 0,C 180,E1 28557.837,E2 28557.837} C_VEL
LIN {X 0,Y 619.263,Z 622.776,A -85,B 0,C 180,E1 28556.846,E2 28556.846} C_VEL
LIN {X 0,Y 618.58,Z 645.235,A -85,B 0,C 180,E1 28556.311,E2 28556.311} C_VEL
LIN {X 0,Y 617.745,Z 666.569,A -85,B 0,C 180,E1 28555.635,E2 28555.635} C_VEL
LIN {X 0,Y 616.764,Z 688.482,A -85,B 0,C 180,E1 28554.761,E2 28554.761} C_VEL
LIN {X 0,Y 615.723,Z 709.232,A -85,B 0,C 180,E1 28553.749,E2 28553.749} C_VEL
LIN {X 0,Y 614.65,Z 728.503,A -85,B 0,C 180,E1 28552.622,E2 28552.622} C_VEL
LIN {X 0,Y 613.531,Z 747.331,A -85,B 0,C 180,E1 28551.311,E2 28551.311} C_VEL
LIN {X 0,Y 612.467,Z 763.817,A -85,B 0,C 180,E1 28549.95,E2 28549.95} C_VEL
LIN {X 0,Y 611.501,Z 778.996,A -85,B 0,C 180,E1 28548.488,E2 28548.488} C_VEL
LIN {X 0,Y 610.622,Z 792.738,A -85,B 0,C 180,E1 28546.946,E2 28546.946} C_VEL
LIN {X 0,Y 609.856,Z 805.133,A -85,B 0,C 180,E1 28545.306,E2 28545.306} C_VEL
LIN {X 0,Y 609.223,Z 816.24,A -85,B 0,C 180,E1 28543.574,E2 28543.574} C_VEL
LIN {X 0,Y 608.735,Z 826.087,A -85,B 0,C 180,E1 28541.752,E2 28541.752} C_VEL
LIN {X 0,Y 608.374,Z 834.479,A -85,B 0,C 180,E1 28539.842,E2 28539.842} C_VEL
LIN {X 0,Y 608.146,Z 841.105,A -85,B 0,C 180,E1 28537.939,E2 28537.939} C_VEL
LIN {X 0,Y 608.04,Z 846.258,A -85,B 0,C 180,E1 28536.041,E2 28536.041} C_VEL
LIN {X 0,Y 607.974,Z 850.366,A -85,B 0,C 180,E1 28533.866,E2 28533.866} C_VEL
LIN {X 0,Y 607.953,Z 852.525,A -85,B 0,C 180,E1 28531.791,E2 28531.791} C_VEL
LIN {X 0,Y 607.944,Z 853.145,A -85,B 0,C 180,E1 28529.812,E2 28529.812} C_VEL
LIN {X 0,Y 607.95,Z 852.331,A -85,B 0,C 180,E1 28527.832,E2 28527.832} C_VEL
LIN {X 0,Y 607.989,Z 849.591,A -85,B 0,C 180,E1 28525.567,E2 28525.567} C_VEL
LIN {X 0,Y 608.058,Z 845.335,A -85,B 0,C 180,E1 28523.485,E2 28523.485} C_VEL
LIN {X 0,Y 608.207,Z 839.338,A -85,B 0,C 180,E1 28521.396,E2 28521.396} C_VEL
LIN {X 0,Y 608.498,Z 831.712,A -85,B 0,C 180,E1 28519.395,E2 28519.395} C_VEL
LIN {X 0,Y 608.887,Z 822.613,A -85,B 0,C 180,E1 28517.481,E2 28517.481} C_VEL
LIN {X 0,Y 609.443,Z 812.13,A -85,B 0,C 180,E1 28515.656,E2 28515.656} C_VEL
LIN {X 0,Y 610.158,Z 800.248,A -85,B 0,C 180,E1 28513.922,E2 28513.922} C_VEL
LIN {X 0,Y 611.004,Z 786.675,A -85,B 0,C 180,E1 28512.257,E2 28512.257} C_VEL
LIN {X 0,Y 611.971,Z 771.582,A -85,B 0,C 180,E1 28510.679,E2 28510.679} C_VEL
LIN {X 0,Y 612.988,Z 755.781,A -85,B 0,C 180,E1 28509.27,E2 28509.27} C_VEL
LIN {X 0,Y 614.111,Z 737.807,A -85,B 0,C 180,E1 28507.907,E2 28507.907} C_VEL
LIN {X 0,Y 615.156,Z 719.448,A -85,B 0,C 180,E1 28506.735,E2 28506.735} C_VEL
LIN {X 0,Y 616.177,Z 700.451,A -85,B 0,C 180,E1 28505.71,E2 28505.71} C_VEL
LIN {X 0,Y 617.171,Z 679.815,A -85,B 0,C 180,E1 28504.78,E2 28504.78} C_VEL
LIN {X 0,Y 618.091,Z 658.548,A -85,B 0,C 180,E1 28503.998,E2 28503.998} C_VEL
LIN {X 0,Y 618.873,Z 636.219,A -85,B 0,C 180,E1 28503.362,E2 28503.362} C_VEL
LIN {X 0,Y 619.458,Z 614.138,A -85,B 0,C 180,E1 28502.91,E2 28502.91} C_VEL
LIN {X 0,Y 623.142,Z 469.818,A -85,B 0,C 180,E1 28500.734,E2 28500.734} C_VEL
LIN {X 0,Y 625.193,Z 372.412,A -85,B 0,C 180,E1 28499.412,E2 28499.412} C_VEL
LIN {X 0,Y 625.761,Z 329.323,A -85,B 0,C 180,E1 28498.848,E2 28498.848} C_VEL
LIN {X 0,Y 625.683,Z 301.876,A -85,B 0,C 180,E1 28497.034,E2 28497.034} C_VEL
LIN {X 0,Y 626.834,Z 263.084,A -85,B 0,C 180,E1 28494.224,E2 28494.224} C_VEL
LIN {X 0,Y 627.148,Z 254.032,A -85,B 0,C 180,E1 28493.561,E2 28493.561} C_VEL
LIN {X 0,Y 619.261,Z 233.33,A -85,B 0,C 180,E1 28491.446,E2 28491.446} C_VEL
LIN {X 0,Y 611.939,Z 216.296,A -85,B 0,C 180,E1 28489.735,E2 28489.735} C_VEL
LIN {X 0,Y 609.278,Z 210.504,A -85,B 0,C 180,E1 28489.161,E2 28489.161} C_VEL
LIN {X 0,Y 609.046,Z 209.357,A -85,B 0,C 180,E1 28489.043,E2 28489.043} C_VEL
LIN {X 0,Y 609.071,Z 209.359,A -85,B 0,C 180,E1 28485.888,E2 28485.888} C_VEL
LIN {X 0,Y 609.052,Z 209.361,A -85,B 0,C 180,E1 28482.69,E2 28482.69} C_VEL
LIN {X 0,Y 609.076,Z 209.359,A -85,B 0,C 180,E1 28479.444,E2 28479.444} C_VEL
LIN {X 0,Y 609.07,Z 209.355,A -85,B 0,C 180,E1 28476.128,E2 28476.128} C_VEL
LIN {X 0,Y 609.053,Z 209.349,A -85,B 0,C 180,E1 28472.916,E2 28472.916} C_VEL
LIN {X 0,Y 609.064,Z 209.355,A -85,B 0,C 180,E1 28469.83,E2 28469.83} C_VEL
LIN {X 0,Y 609.061,Z 209.358,A -85,B 0,C 180,E1 28466.627,E2 28466.627} C_VEL
LIN {X 0,Y 609.069,Z 209.339,A -85,B 0,C 180,E1 28463.409,E2 28463.409} C_VEL
LIN {X 0,Y 609.069,Z 209.357,A -85,B 0,C 180,E1 28460.11,E2 28460.11} C_VEL
LIN {X 0,Y 609.061,Z 209.347,A -85,B 0,C 180,E1 28456.842,E2 28456.842} C_VEL
LIN {X 0,Y 609.056,Z 209.35,A -85,B 0,C 180,E1 28453.771,E2 28453.771} C_VEL
LIN {X 0,Y 609.064,Z 209.35,A -85,B 0,C 180,E1 28450.595,E2 28450.595} C_VEL
LIN {X 0,Y 609.055,Z 209.35,A -85,B 0,C 180,E1 28447.435,E2 28447.435} C_VEL
LIN {X 0,Y 609.068,Z 209.354,A -85,B 0,C 180,E1 28444.142,E2 28444.142} C_VEL
LIN {X 0,Y 609.075,Z 209.352,A -85,B 0,C 180,E1 28440.941,E2 28440.941} C_VEL
LIN {X 0,Y 609.049,Z 209.36,A -85,B 0,C 180,E1 28437.742,E2 28437.742} C_VEL
LIN {X 0,Y 609.07,Z 209.357,A -85,B 0,C 180,E1 28434.536,E2 28434.536} C_VEL
LIN {X 0,Y 609.043,Z 209.355,A -85,B 0,C 180,E1 28431.408,E2 28431.408} C_VEL
LIN {X 0,Y 609.073,Z 209.365,A -85,B 0,C 180,E1 28428.158,E2 28428.158} C_VEL
LIN {X 0,Y 609.06,Z 209.357,A -85,B 0,C 180,E1 28424.966,E2 28424.966} C_VEL
LIN {X 0,Y 609.045,Z 209.36,A -85,B 0,C 180,E1 28421.725,E2 28421.725} C_VEL
LIN {X 0,Y 609.077,Z 209.358,A -85,B 0,C 180,E1 28418.562,E2 28418.562} C_VEL
LIN {X 0,Y 609.035,Z 209.363,A -85,B 0,C 180,E1 28415.441,E2 28415.441} C_VEL
LIN {X 0,Y 609.076,Z 209.359,A -85,B 0,C 180,E1 28412.316,E2 28412.316} C_VEL
LIN {X 0,Y 609.031,Z 209.365,A -85,B 0,C 180,E1 28409.297,E2 28409.297} C_VEL
LIN {X 0,Y 609.076,Z 209.358,A -85,B 0,C 180,E1 28406.168,E2 28406.168} C_VEL
LIN {X 0,Y 609.033,Z 209.365,A -85,B 0,C 180,E1 28403.066,E2 28403.066} C_VEL
LIN {X 0,Y 609.048,Z 209.36,A -85,B 0,C 180,E1 28399.819,E2 28399.819} C_VEL
LIN {X 0,Y 609.081,Z 209.513,A -85,B 0,C 180,E1 28397.949,E2 28397.949} C_VEL
LIN {X 0,Y 610.077,Z 212.43,A -85,B 0,C 180,E1 28397.653,E2 28397.653} C_VEL
LIN {X 0,Y 611.359,Z 214.646,A -85,B 0,C 180,E1 28397.382,E2 28397.382} C_VEL
LIN {X 0,Y 622.163,Z 236.027,A -85,B 0,C 180,E1 28394.998,E2 28394.998} C_VEL
LIN {X 0,Y 632.92,Z 258.196,A -85,B 0,C 180,E1 28392.725,E2 28392.725} C_VEL
LIN {X 0,Y 634.211,Z 261.306,A -85,B 0,C 180,E1 28392.437,E2 28392.437} C_VEL
LIN {X 0,Y 631.23,Z 306.025,A -85,B 0,C 180,E1 28390.061,E2 28390.061} C_VEL
LIN {X 0,Y 633.831,Z 325.862,A -85,B 0,C 180,E1 28389.598,E2 28389.598} C_VEL
LIN {X 0,Y 629.969,Z 550.131,A -85,B 0,C 180,E1 28386.667,E2 28386.667} C_VEL
LIN {X 0,Y 627.801,Z 692.847,A -85,B 0,C 180,E1 28384.843,E2 28384.843} C_VEL
LIN {X 0,Y 626.927,Z 717.852,A -85,B 0,C 180,E1 28384.363,E2 28384.363} C_VEL
LIN {X 0,Y 625.933,Z 739.401,A -85,B 0,C 180,E1 28383.812,E2 28383.812} C_VEL
LIN {X 0,Y 624.507,Z 764.89,A -85,B 0,C 180,E1 28382.982,E2 28382.982} C_VEL
LIN {X 0,Y 623.063,Z 787.478,A -85,B 0,C 180,E1 28382.077,E2 28382.077} C_VEL
LIN {X 0,Y 621.444,Z 810.737,A -85,B 0,C 180,E1 28380.953,E2 28380.953} C_VEL
LIN {X 0,Y 619.86,Z 831.434,A -85,B 0,C 180,E1 28379.791,E2 28379.791} C_VEL
LIN {X 0,Y 618.139,Z 852.729,A -85,B 0,C 180,E1 28378.396,E2 28378.396} C_VEL
LIN {X 0,Y 616.56,Z 872.034,A -85,B 0,C 180,E1 28376.954,E2 28376.954} C_VEL
LIN {X 0,Y 614.929,Z 891.256,A -85,B 0,C 180,E1 28375.301,E2 28375.301} C_VEL
LIN {X 0,Y 613.765,Z 905.347,A -85,B 0,C 180,E1 28373.932,E2 28373.932} C_VEL
LIN {X 0,Y 612.386,Z 920.985,A -85,B 0,C 180,E1 28372.159,E2 28372.159} C_VEL
LIN {X 0,Y 611.099,Z 935.912,A -85,B 0,C 180,E1 28370.197,E2 28370.197} C_VEL
LIN {X 0,Y 610.065,Z 949.661,A -85,B 0,C 180,E1 28368.144,E2 28368.144} C_VEL
LIN {X 0,Y 609.286,Z 961.309,A -85,B 0,C 180,E1 28366.102,E2 28366.102} C_VEL
LIN {X 0,Y 608.741,Z 971.393,A -85,B 0,C 180,E1 28364.069,E2 28364.069} C_VEL
LIN {X 0,Y 608.345,Z 980.543,A -85,B 0,C 180,E1 28361.856,E2 28361.856} C_VEL
LIN {X 0,Y 608.116,Z 987.422,A -85,B 0,C 180,E1 28359.846,E2 28359.846} C_VEL
LIN {X 0,Y 607.957,Z 993.863,A -85,B 0,C 180,E1 28357.465,E2 28357.465} C_VEL
LIN {X 0,Y 607.909,Z 997.814,A -85,B 0,C 180,E1 28355.474,E2 28355.474} C_VEL
LIN {X 0,Y 607.905,Z 1000.689,A -85,B 0,C 180,E1 28353.395,E2 28353.395} C_VEL
LIN {X 0,Y 607.902,Z 1002.259,A -85,B 0,C 180,E1 28351.037,E2 28351.037} C_VEL
LIN {X 0,Y 607.89,Z 1002.304,A -85,B 0,C 180,E1 28349.152,E2 28349.152} C_VEL
LIN {X 0,Y 607.887,Z 1001.087,A -85,B 0,C 180,E1 28346.983,E2 28346.983} C_VEL
LIN {X 0,Y 607.903,Z 998.132,A -85,B 0,C 180,E1 28344.715,E2 28344.715} C_VEL
LIN {X 0,Y 607.963,Z 994.482,A -85,B 0,C 180,E1 28342.82,E2 28342.82} C_VEL
LIN {X 0,Y 608.096,Z 988.633,A -85,B 0,C 180,E1 28340.536,E2 28340.536} C_VEL
LIN {X 0,Y 608.289,Z 981.6,A -85,B 0,C 180,E1 28338.431,E2 28338.431} C_VEL
LIN {X 0,Y 608.632,Z 973.534,A -85,B 0,C 180,E1 28336.413,E2 28336.413} C_VEL
LIN {X 0,Y 609.198,Z 962.857,A -85,B 0,C 180,E1 28334.189,E2 28334.189} C_VEL
LIN {X 0,Y 609.898,Z 952.127,A -85,B 0,C 180,E1 28332.273,E2 28332.273} C_VEL
LIN {X 0,Y 610.945,Z 938.013,A -85,B 0,C 180,E1 28330.098,E2 28330.098} C_VEL
LIN {X 0,Y 612.012,Z 924.841,A -85,B 0,C 180,E1 28328.332,E2 28328.332} C_VEL
LIN {X 0,Y 613.526,Z 908.15,A -85,B 0,C 180,E1 28326.364,E2 28326.364} C_VEL
LIN {X 0,Y 614.591,Z 895.26,A -85,B 0,C 180,E1 28325.079,E2 28325.079} C_VEL
LIN {X 0,Y 615.854,Z 878.985,A -85,B 0,C 180,E1 28323.666,E2 28323.666} C_VEL
LIN {X 0,Y 617.384,Z 859.422,A -85,B 0,C 180,E1 28322.164,E2 28322.164} C_VEL
LIN {X 0,Y 618.881,Z 838.77,A -85,B 0,C 180,E1 28320.796,E2 28320.796} C_VEL
LIN {X 0,Y 620.437,Z 816.025,A -85,B 0,C 180,E1 28319.492,E2 28319.492} C_VEL
LIN {X 0,Y 621.785,Z 794.8,A -85,B 0,C 180,E1 28318.462,E2 28318.462} C_VEL
LIN {X 0,Y 623.109,Z 770.964,A -85,B 0,C 180,E1 28317.482,E2 28317.482} C_VEL
LIN {X 0,Y 624.156,Z 748.988,A -85,B 0,C 180,E1 28316.745,E2 28316.745} C_VEL
LIN {X 0,Y 625.146,Z 724.43,A -85,B 0,C 180,E1 28316.083,E2 28316.083} C_VEL
LIN {X 0,Y 625.847,Z 701.437,A -85,B 0,C 180,E1 28315.625,E2 28315.625} C_VEL
LIN {X 0,Y 626.312,Z 674.817,A -85,B 0,C 180,E1 28315.252,E2 28315.252} C_VEL
LIN {X 0,Y 627.717,Z 491.439,A -85,B 0,C 180,E1 28313.094,E2 28313.094} C_VEL
LIN {X 0,Y 629.694,Z 341.468,A -85,B 0,C 180,E1 28311.173,E2 28311.173} C_VEL
LIN {X 0,Y 629.797,Z 322.462,A -85,B 0,C 180,E1 28310.901,E2 28310.901} C_VEL
LIN {X 0,Y 628.881,Z 316.063,A -85,B 0,C 180,E1 28310.743,E2 28310.743} C_VEL
LIN {X 0,Y 632.1,Z 287.734,A -85,B 0,C 180,E1 28309.029,E2 28309.029} C_VEL
LIN {X 0,Y 636.352,Z 263.054,A -85,B 0,C 180,E1 28307.388,E2 28307.388} C_VEL
LIN {X 0,Y 633.88,Z 255.73,A -85,B 0,C 180,E1 28306.258,E2 28306.258} C_VEL
LIN {X 0,Y 631.684,Z 249.812,A -85,B 0,C 180,E1 28305.037,E2 28305.037} C_VEL
LIN {X 0,Y 630.151,Z 246.148,A -85,B 0,C 180,E1 28303.914,E2 28303.914} C_VEL
LIN {X 0,Y 629.209,Z 243.68,A -85,B 0,C 180,E1 28302.607,E2 28302.607} C_VEL
LIN {X 0,Y 629.197,Z 242.962,A -85,B 0,C 180,E1 28301.677,E2 28301.677} C_VEL
LIN {X 0,Y 629.247,Z 244.845,A -85,B 0,C 180,E1 28300.294,E2 28300.294} C_VEL
LIN {X 0,Y 630.015,Z 246.442,A -85,B 0,C 180,E1 28299.526,E2 28299.526} C_VEL
LIN {X 0,Y 631.27,Z 250.62,A -85,B 0,C 180,E1 28298.367,E2 28298.367} C_VEL
LIN {X 0,Y 633.282,Z 257.321,A -85,B 0,C 180,E1 28297.055,E2 28297.055} C_VEL
LIN {X 0,Y 633.886,Z 259.837,A -85,B 0,C 180,E1 28296.659,E2 28296.659} C_VEL
LIN {X 0,Y 628.956,Z 286.56,A -85,B 0,C 180,E1 28294.524,E2 28294.524} C_VEL
LIN {X 0,Y 624.452,Z 322.133,A -85,B 0,C 180,E1 28291.898,E2 28291.898} C_VEL
LIN {X 0,Y 620.823,Z 364.601,A -85,B 0,C 180,E1 28288.946,E2 28288.946} C_VEL
LIN {X 0,Y 617.801,Z 412.201,A -85,B 0,C 180,E1 28285.809,E2 28285.809} C_VEL
LIN {X 0,Y 616.724,Z 435.374,A -85,B 0,C 180,E1 28284.347,E2 28284.347} C_VEL
LIN {X 0,Y 620.799,Z 471.664,A -85,B 0,C 180,E1 28283.283,E2 28283.283} C_VEL
LIN {X 0,Y 622.255,Z 490.045,A -85,B 0,C 180,E1 28282.818,E2 28282.818} C_VEL
LIN {X 0,Y 617.805,Z 602.169,A -85,B 0,C 180,E1 28280.908,E2 28280.908} C_VEL
LIN {X 0,Y 615.556,Z 685.269,A -85,B 0,C 180,E1 28279.561,E2 28279.561} C_VEL
LIN {X 0,Y 614.874,Z 706.996,A -85,B 0,C 180,E1 28279.026,E2 28279.026} C_VEL
LIN {X 0,Y 614.2,Z 726.92,A -85,B 0,C 180,E1 28278.359,E2 28278.359} C_VEL
LIN {X 0,Y 613.468,Z 745.927,A -85,B 0,C 180,E1 28277.543,E2 28277.543} C_VEL
LIN {X 0,Y 612.789,Z 762.834,A -85,B 0,C 180,E1 28276.64,E2 28276.64} C_VEL
LIN {X 0,Y 612.093,Z 779.124,A -85,B 0,C 180,E1 28275.588,E2 28275.588} C_VEL
LIN {X 0,Y 611.422,Z 793.892,A -85,B 0,C 180,E1 28274.442,E2 28274.442} C_VEL
LIN {X 0,Y 610.824,Z 806.763,A -85,B 0,C 180,E1 28273.248,E2 28273.248} C_VEL
LIN {X 0,Y 610.268,Z 818.84,A -85,B 0,C 180,E1 28271.914,E2 28271.914} C_VEL
LIN {X 0,Y 609.752,Z 830.204,A -85,B 0,C 180,E1 28270.392,E2 28270.392} C_VEL
LIN {X 0,Y 609.35,Z 839.415,A -85,B 0,C 180,E1 28268.873,E2 28268.873} C_VEL
LIN {X 0,Y 609.04,Z 847.181,A -85,B 0,C 180,E1 28267.262,E2 28267.262} C_VEL
LIN {X 0,Y 608.824,Z 853.415,A -85,B 0,C 180,E1 28265.561,E2 28265.561} C_VEL
LIN {X 0,Y 608.661,Z 857.803,A -85,B 0,C 180,E1 28263.862,E2 28263.862} C_VEL
LIN {X 0,Y 608.554,Z 860.573,A -85,B 0,C 180,E1 28262.072,E2 28262.072} C_VEL
LIN {X 0,Y 608.499,Z 861.523,A -85,B 0,C 180,E1 28260.282,E2 28260.282} C_VEL
LIN {X 0,Y 608.468,Z 860.678,A -85,B 0,C 180,E1 28258.493,E2 28258.493} C_VEL
LIN {X 0,Y 608.485,Z 858.041,A -85,B 0,C 180,E1 28256.703,E2 28256.703} C_VEL
LIN {X 0,Y 608.548,Z 853.835,A -85,B 0,C 180,E1 28255.004,E2 28255.004} C_VEL
LIN {X 0,Y 608.676,Z 847.868,A -85,B 0,C 180,E1 28253.302,E2 28253.302} C_VEL
LIN {X 0,Y 608.9,Z 839.974,A -85,B 0,C 180,E1 28251.596,E2 28251.596} C_VEL
LIN {X 0,Y 609.235,Z 830.491,A -85,B 0,C 180,E1 28249.976,E2 28249.976} C_VEL
LIN {X 0,Y 609.671,Z 819.569,A -85,B 0,C 180,E1 28248.458,E2 28248.458} C_VEL
LIN {X 0,Y 610.207,Z 807.122,A -85,B 0,C 180,E1 28247.027,E2 28247.027} C_VEL
LIN {X 0,Y 610.844,Z 793.148,A -85,B 0,C 180,E1 28245.69,E2 28245.69} C_VEL
LIN {X 0,Y 611.562,Z 777.487,A -85,B 0,C 180,E1 28244.447,E2 28244.447} C_VEL
LIN {X 0,Y 612.301,Z 760.669,A -85,B 0,C 180,E1 28243.346,E2 28243.346} C_VEL
LIN {X 0,Y 613.009,Z 743.732,A -85,B 0,C 180,E1 28242.437,E2 28242.437} C_VEL
LIN {X 0,Y 613.709,Z 726.099,A -85,B 0,C 180,E1 28241.672,E2 28241.672} C_VEL
LIN {X 0,Y 614.339,Z 706.874,A -85,B 0,C 180,E1 28241.025,E2 28241.025} C_VEL
LIN {X 0,Y 614.884,Z 687.11,A -85,B 0,C 180,E1 28240.543,E2 28240.543} C_VEL
LIN {X 0,Y 615.326,Z 663.198,A -85,B 0,C 180,E1 28240.169,E2 28240.169} C_VEL
LIN {X 0,Y 618.192,Z 485.565,A -85,B 0,C 180,E1 28237.744,E2 28237.744} C_VEL
LIN {X 0,Y 615.087,Z 459.086,A -85,B 0,C 180,E1 28237.211,E2 28237.211} C_VEL
LIN {X 0,Y 617.03,Z 406.969,A -85,B 0,C 180,E1 28234.017,E2 28234.017} C_VEL
LIN {X 0,Y 619.24,Z 355.289,A -85,B 0,C 180,E1 28230.814,E2 28230.814} C_VEL
LIN {X 0,Y 619.749,Z 343.494,A -85,B 0,C 180,E1 28230.076,E2 28230.076} C_VEL
LIN {X 0,Y 619.14,Z 337.327,A -85,B 0,C 180,E1 28229.644,E2 28229.644} C_VEL
LIN {X 0,Y 614.246,Z 321.833,A -85,B 0,C 180,E1 28228.37,E2 28228.37} C_VEL
LIN {X 0,Y 613.838,Z 316.525,A -85,B 0,C 180,E1 28227.995,E2 28227.995} C_VEL
LIN {X 0,Y 616.449,Z 266.722,A -85,B 0,C 180,E1 28224.786,E2 28224.786} C_VEL
LIN {X 0,Y 617.09,Z 251.696,A -85,B 0,C 180,E1 28223.797,E2 28223.797} C_VEL
LIN {X 0,Y 607.428,Z 226.45,A -85,B 0,C 180,E1 28221.4,E2 28221.4} C_VEL
LIN {X 0,Y 601.069,Z 210.359,A -85,B 0,C 180,E1 28219.779,E2 28219.779} C_VEL
LIN {X 0,Y 601.14,Z 210.349,A -85,B 0,C 180,E1 28216.741,E2 28216.741} C_VEL
LIN {X 0,Y 601.131,Z 210.351,A -85,B 0,C 180,E1 28213.512,E2 28213.512} C_VEL
LIN {X 0,Y 601.107,Z 210.401,A -85,B 0,C 180,E1 28211.392,E2 28211.392} C_VEL
LIN {X 0,Y 602.316,Z 213.709,A -85,B 0,C 180,E1 28211.09,E2 28211.09} C_VEL
LIN {X 0,Y 609.678,Z 230.052,A -85,B 0,C 180,E1 28209.425,E2 28209.425} C_VEL
LIN {X 0,Y 616.94,Z 248.368,A -85,B 0,C 180,E1 28207.546,E2 28207.546} C_VEL
LIN {X 0,Y 620.346,Z 257.325,A -85,B 0,C 180,E1 28206.611,E2 28206.611} C_VEL
LIN {X 0,Y 619.056,Z 301.971,A -85,B 0,C 180,E1 28203.378,E2 28203.378} C_VEL
LIN {X 0,Y 619.115,Z 330.54,A -85,B 0,C 180,E1 28201.489,E2 28201.489} C_VEL
LIN {X 0,Y 619.023,Z 333.002,A -85,B 0,C 180,E1 28201.386,E2 28201.386} C_VEL
LIN {X 0,Y 617.053,Z 436.465,A -85,B 0,C 180,E1 28200.024,E2 28200.024} C_VEL
LIN {X 0,Y 614.006,Z 548.9,A -85,B 0,C 180,E1 28198.353,E2 28198.353} C_VEL
LIN {X 0,Y 611.96,Z 623.565,A -85,B 0,C 180,E1 28197.142,E2 28197.142} C_VEL
LIN {X 0,Y 611.256,Z 645.434,A -85,B 0,C 180,E1 28196.613,E2 28196.613} C_VEL
LIN {X 0,Y 610.36,Z 666.913,A -85,B 0,C 180,E1 28195.924,E2 28195.924} C_VEL
LIN {X 0,Y 609.344,Z 688.042,A -85,B 0,C 180,E1 28195.069,E2 28195.069} C_VEL
LIN {X 0,Y 608.275,Z 707.568,A -85,B 0,C 180,E1 28194.11,E2 28194.11} C_VEL
LIN {X 0,Y 607.029,Z 728.422,A -85,B 0,C 180,E1 28192.876,E2 28192.876} C_VEL
LIN {X 0,Y 605.838,Z 747.388,A -85,B 0,C 180,E1 28191.544,E2 28191.544} C_VEL
LIN {X 0,Y 604.738,Z 764.055,A -85,B 0,C 180,E1 28190.166,E2 28190.166} C_VEL
LIN {X 0,Y 603.705,Z 779.814,A -85,B 0,C 180,E1 28188.642,E2 28188.642} C_VEL
LIN {X 0,Y 602.798,Z 793.738,A -85,B 0,C 180,E1 28187.074,E2 28187.074} C_VEL
LIN {X 0,Y 602.008,Z 806.213,A -85,B 0,C 180,E1 28185.411,E2 28185.411} C_VEL
LIN {X 0,Y 601.348,Z 817.34,A -85,B 0,C 180,E1 28183.657,E2 28183.657} C_VEL
LIN {X 0,Y 600.838,Z 827.201,A -85,B 0,C 180,E1 28181.812,E2 28181.812} C_VEL
LIN {X 0,Y 600.475,Z 835.217,A -85,B 0,C 180,E1 28179.973,E2 28179.973} C_VEL
LIN {X 0,Y 600.224,Z 842.262,A -85,B 0,C 180,E1 28177.948,E2 28177.948} C_VEL
LIN {X 0,Y 600.103,Z 847.613,A -85,B 0,C 180,E1 28175.93,E2 28175.93} C_VEL
LIN {X 0,Y 600.037,Z 851.301,A -85,B 0,C 180,E1 28173.918,E2 28173.918} C_VEL
LIN {X 0,Y 600.016,Z 853.513,A -85,B 0,C 180,E1 28171.814,E2 28171.814} C_VEL
LIN {X 0,Y 600.006,Z 854.165,A -85,B 0,C 180,E1 28169.714,E2 28169.714} C_VEL
LIN {X 0,Y 600.012,Z 853.186,A -85,B 0,C 180,E1 28167.612,E2 28167.612} C_VEL
LIN {X 0,Y 600.052,Z 850.676,A -85,B 0,C 180,E1 28165.604,E2 28165.604} C_VEL
LIN {X 0,Y 600.131,Z 846.465,A -85,B 0,C 180,E1 28163.495,E2 28163.495} C_VEL
LIN {X 0,Y 600.284,Z 840.789,A -85,B 0,C 180,E1 28161.475,E2 28161.475} C_VEL
LIN {X 0,Y 600.569,Z 833.231,A -85,B 0,C 180,E1 28159.447,E2 28159.447} C_VEL
LIN {X 0,Y 600.973,Z 824.228,A -85,B 0,C 180,E1 28157.509,E2 28157.509} C_VEL
LIN {X 0,Y 601.547,Z 813.84,A -85,B 0,C 180,E1 28155.661,E2 28155.661} C_VEL
LIN {X 0,Y 602.272,Z 801.989,A -85,B 0,C 180,E1 28153.904,E2 28153.904} C_VEL
LIN {X 0,Y 603.118,Z 788.653,A -85,B 0,C 180,E1 28152.239,E2 28152.239} C_VEL
LIN {X 0,Y 604.152,Z 772.909,A -85,B 0,C 180,E1 28150.57,E2 28150.57} C_VEL
LIN {X 0,Y 605.205,Z 757.135,A -85,B 0,C 180,E1 28149.143,E2 28149.143} C_VEL
LIN {X 0,Y 606.362,Z 739.202,A -85,B 0,C 180,E1 28147.763,E2 28147.763} C_VEL
LIN {X 0,Y 607.618,Z 718.665,A -85,B 0,C 180,E1 28146.429,E2 28146.429} C_VEL
LIN {X 0,Y 608.767,Z 698.662,A -85,B 0,C 180,E1 28145.343,E2 28145.343} C_VEL
LIN {X 0,Y 609.835,Z 678.194,A -85,B 0,C 180,E1 28144.42,E2 28144.42} C_VEL
LIN {X 0,Y 610.848,Z 655.983,A -85,B 0,C 180,E1 28143.614,E2 28143.614} C_VEL
LIN {X 0,Y 611.622,Z 634.616,A -85,B 0,C 180,E1 28143.014,E2 28143.014} C_VEL
LIN {X 0,Y 612.258,Z 612.134,A -85,B 0,C 180,E1 28142.558,E2 28142.558} C_VEL
LIN {X 0,Y 616.092,Z 474.409,A -85,B 0,C 180,E1 28140.429,E2 28140.429} C_VEL
LIN {X 0,Y 618.233,Z 380.383,A -85,B 0,C 180,E1 28139.128,E2 28139.128} C_VEL
LIN {X 0,Y 619.158,Z 331.734,A -85,B 0,C 180,E1 28138.491,E2 28138.491} C_VEL
LIN {X 0,Y 619.032,Z 304.277,A -85,B 0,C 180,E1 28136.689,E2 28136.689} C_VEL
LIN {X 0,Y 620.167,Z 264.814,A -85,B 0,C 180,E1 28133.836,E2 28133.836} C_VEL
LIN {X 0,Y 620.21,Z 257,A -85,B 0,C 180,E1 28133.25,E2 28133.25} C_VEL
LIN {X 0,Y 612.431,Z 236.635,A -85,B 0,C 180,E1 28131.149,E2 28131.149} C_VEL
LIN {X 0,Y 604.446,Z 218.015,A -85,B 0,C 180,E1 28129.257,E2 28129.257} C_VEL
LIN {X 0,Y 601.233,Z 211.02,A -85,B 0,C 180,E1 28128.555,E2 28128.555} C_VEL
LIN {X 0,Y 601.127,Z 210.345,A -85,B 0,C 180,E1 28128.462,E2 28128.462} C_VEL
LIN {X 0,Y 601.116,Z 210.356,A -85,B 0,C 180,E1 28125.148,E2 28125.148} C_VEL
LIN {X 0,Y 601.131,Z 210.356,A -85,B 0,C 180,E1 28121.965,E2 28121.965} C_VEL
LIN {X 0,Y 601.114,Z 210.353,A -85,B 0,C 180,E1 28118.837,E2 28118.837} C_VEL
LIN {X 0,Y 601.131,Z 210.349,A -85,B 0,C 180,E1 28115.604,E2 28115.604} C_VEL
LIN {X 0,Y 601.129,Z 210.338,A -85,B 0,C 180,E1 28112.33,E2 28112.33} C_VEL
LIN {X 0,Y 601.123,Z 210.341,A -85,B 0,C 180,E1 28109.059,E2 28109.059} C_VEL
LIN {X 0,Y 601.125,Z 210.349,A -85,B 0,C 180,E1 28105.836,E2 28105.836} C_VEL
LIN {X 0,Y 601.119,Z 210.333,A -85,B 0,C 180,E1 28102.597,E2 28102.597} C_VEL
LIN {X 0,Y 601.127,Z 210.338,A -85,B 0,C 180,E1 28099.417,E2 28099.417} C_VEL
LIN {X 0,Y 601.132,Z 210.346,A -85,B 0,C 180,E1 28096.128,E2 28096.128} C_VEL
LIN {X 0,Y 601.127,Z 210.333,A -85,B 0,C 180,E1 28092.879,E2 28092.879} C_VEL
LIN {X 0,Y 601.115,Z 210.351,A -85,B 0,C 180,E1 28089.672,E2 28089.672} C_VEL
LIN {X 0,Y 601.126,Z 210.33,A -85,B 0,C 180,E1 28086.495,E2 28086.495} C_VEL
LIN {X 0,Y 601.122,Z 210.347,A -85,B 0,C 180,E1 28083.242,E2 28083.242} C_VEL
LIN {X 0,Y 601.116,Z 210.326,A -85,B 0,C 180,E1 28079.905,E2 28079.905} C_VEL
LIN {X 0,Y 601.131,Z 210.347,A -85,B 0,C 180,E1 28076.663,E2 28076.663} C_VEL
LIN {X 0,Y 601.104,Z 210.328,A -85,B 0,C 180,E1 28073.505,E2 28073.505} C_VEL
LIN {X 0,Y 601.133,Z 210.347,A -85,B 0,C 180,E1 28070.329,E2 28070.329} C_VEL
LIN {X 0,Y 601.117,Z 210.347,A -85,B 0,C 180,E1 28067.096,E2 28067.096} C_VEL
LIN {X 0,Y 601.107,Z 210.355,A -85,B 0,C 180,E1 28063.772,E2 28063.772} C_VEL
LIN {X 0,Y 601.137,Z 210.346,A -85,B 0,C 180,E1 28060.569,E2 28060.569} C_VEL
LIN {X 0,Y 601.097,Z 210.354,A -85,B 0,C 180,E1 28057.4,E2 28057.4} C_VEL
LIN {X 0,Y 601.137,Z 210.354,A -85,B 0,C 180,E1 28054.27,E2 28054.27} C_VEL
LIN {X 0,Y 601.099,Z 210.35,A -85,B 0,C 180,E1 28051.158,E2 28051.158} C_VEL
LIN {X 0,Y 601.122,Z 210.35,A -85,B 0,C 180,E1 28047.953,E2 28047.953} C_VEL
LIN {X 0,Y 601.11,Z 210.352,A -85,B 0,C 180,E1 28044.862,E2 28044.862} C_VEL
LIN {X 0,Y 601.093,Z 210.352,A -85,B 0,C 180,E1 28041.581,E2 28041.581} C_VEL
LIN {X 0,Y 601.149,Z 210.526,A -85,B 0,C 180,E1 28038.641,E2 28038.641} C_VEL
LIN {X 0,Y 602.474,Z 213.87,A -85,B 0,C 180,E1 28038.278,E2 28038.278} C_VEL
LIN {X 0,Y 603.677,Z 216.239,A -85,B 0,C 180,E1 28037.998,E2 28037.998} C_VEL
LIN {X 0,Y 612.281,Z 233.182,A -85,B 0,C 180,E1 28036.048,E2 28036.048} C_VEL
LIN {X 0,Y 623.73,Z 256.375,A -85,B 0,C 180,E1 28033.577,E2 28033.577} C_VEL
LIN {X 0,Y 627.625,Z 264.84,A -85,B 0,C 180,E1 28032.74,E2 28032.74} C_VEL
LIN {X 0,Y 624.68,Z 306.779,A -85,B 0,C 180,E1 28030.491,E2 28030.491} C_VEL
LIN {X 0,Y 627.288,Z 327.204,A -85,B 0,C 180,E1 28030.005,E2 28030.005} C_VEL
LIN {X 0,Y 622.673,Z 577.422,A -85,B 0,C 180,E1 28026.695,E2 28026.695} C_VEL
LIN {X 0,Y 620.808,Z 692.639,A -85,B 0,C 180,E1 28025.205,E2 28025.205} C_VEL
LIN {X 0,Y 619.891,Z 717.552,A -85,B 0,C 180,E1 28024.722,E2 28024.722} C_VEL
LIN {X 0,Y 618.86,Z 738.778,A -85,B 0,C 180,E1 28024.176,E2 28024.176} C_VEL
LIN {X 0,Y 617.374,Z 764.189,A -85,B 0,C 180,E1 28023.342,E2 28023.342} C_VEL
LIN {X 0,Y 615.935,Z 785.11,A -85,B 0,C 180,E1 28022.502,E2 28022.502} C_VEL
LIN {X 0,Y 614.215,Z 808.946,A -85,B 0,C 180,E1 28021.356,E2 28021.356} C_VEL
LIN {X 0,Y 612.615,Z 828.882,A -85,B 0,C 180,E1 28020.233,E2 28020.233} C_VEL
LIN {X 0,Y 610.668,Z 851.586,A -85,B 0,C 180,E1 28018.749,E2 28018.749} C_VEL
LIN {X 0,Y 609.029,Z 870.543,A -85,B 0,C 180,E1 28017.32,E2 28017.32} C_VEL
LIN {X 0,Y 607.278,Z 890.328,A -85,B 0,C 180,E1 28015.608,E2 28015.608} C_VEL
LIN {X 0,Y 605.874,Z 906.64,A -85,B 0,C 180,E1 28014.004,E2 28014.004} C_VEL
LIN {X 0,Y 604.409,Z 923.986,A -85,B 0,C 180,E1 28012.057,E2 28012.057} C_VEL
LIN {X 0,Y 603.355,Z 935.91,A -85,B 0,C 180,E1 28010.467,E2 28010.467} C_VEL
LIN {X 0,Y 602.248,Z 949.662,A -85,B 0,C 180,E1 28008.388,E2 28008.388} C_VEL
LIN {X 0,Y 601.41,Z 961.308,A -85,B 0,C 180,E1 28006.318,E2 28006.318} C_VEL
LIN {X 0,Y 600.821,Z 971.391,A -85,B 0,C 180,E1 28004.259,E2 28004.259} C_VEL
LIN {X 0,Y 600.388,Z 980.543,A -85,B 0,C 180,E1 28002.015,E2 28002.015} C_VEL
LIN {X 0,Y 600.133,Z 987.422,A -85,B 0,C 180,E1 27999.978,E2 27999.978} C_VEL
LIN {X 0,Y 599.961,Z 993.863,A -85,B 0,C 180,E1 27997.566,E2 27997.566} C_VEL
LIN {X 0,Y 599.914,Z 997.814,A -85,B 0,C 180,E1 27995.547,E2 27995.547} C_VEL
LIN {X 0,Y 599.907,Z 1000.69,A -85,B 0,C 180,E1 27993.44,E2 27993.44} C_VEL
LIN {X 0,Y 599.902,Z 1002.258,A -85,B 0,C 180,E1 27991.05,E2 27991.05} C_VEL
LIN {X 0,Y 599.89,Z 1002.304,A -85,B 0,C 180,E1 27989.14,E2 27989.14} C_VEL
LIN {X 0,Y 599.888,Z 1001.086,A -85,B 0,C 180,E1 27986.942,E2 27986.942} C_VEL
LIN {X 0,Y 599.905,Z 998.132,A -85,B 0,C 180,E1 27984.644,E2 27984.644} C_VEL
LIN {X 0,Y 599.962,Z 994.482,A -85,B 0,C 180,E1 27982.723,E2 27982.723} C_VEL
LIN {X 0,Y 600.113,Z 988.633,A -85,B 0,C 180,E1 27980.409,E2 27980.409} C_VEL
LIN {X 0,Y 600.332,Z 981.6,A -85,B 0,C 180,E1 27978.276,E2 27978.276} C_VEL
LIN {X 0,Y 600.696,Z 973.533,A -85,B 0,C 180,E1 27976.23,E2 27976.23} C_VEL
LIN {X 0,Y 601.309,Z 962.843,A -85,B 0,C 180,E1 27973.974,E2 27973.974} C_VEL
LIN {X 0,Y 602.029,Z 952.538,A -85,B 0,C 180,E1 27972.106,E2 27972.106} C_VEL
LIN {X 0,Y 603.139,Z 938.712,A -85,B 0,C 180,E1 27969.93,E2 27969.93} C_VEL
LIN {X 0,Y 604.242,Z 925.857,A -85,B 0,C 180,E1 27968.177,E2 27968.177} C_VEL
LIN {X 0,Y 605.106,Z 915.265,A -85,B 0,C 180,E1 27966.944,E2 27966.944} C_VEL
LIN {X 0,Y 606.516,Z 898.257,A -85,B 0,C 180,E1 27965.193,E2 27965.193} C_VEL
LIN {X 0,Y 608.005,Z 879.617,A -85,B 0,C 180,E1 27963.534,E2 27963.534} C_VEL
LIN {X 0,Y 609.641,Z 859.612,A -85,B 0,C 180,E1 27961.968,E2 27961.968} C_VEL
LIN {X 0,Y 611.205,Z 838.818,A -85,B 0,C 180,E1 27960.572,E2 27960.572} C_VEL
LIN {X 0,Y 612.789,Z 816.849,A -85,B 0,C 180,E1 27959.288,E2 27959.288} C_VEL
LIN {X 0,Y 614.229,Z 795.108,A -85,B 0,C 180,E1 27958.217,E2 27958.217} C_VEL
LIN {X 0,Y 615.576,Z 772.242,A -85,B 0,C 180,E1 27957.255,E2 27957.255} C_VEL
LIN {X 0,Y 616.728,Z 749.003,A -85,B 0,C 180,E1 27956.464,E2 27956.464} C_VEL
LIN {X 0,Y 617.781,Z 724.379,A -85,B 0,C 180,E1 27955.792,E2 27955.792} C_VEL
LIN {X 0,Y 618.516,Z 701.498,A -85,B 0,C 180,E1 27955.328,E2 27955.328} C_VEL
LIN {X 0,Y 619.007,Z 675.506,A -85,B 0,C 180,E1 27954.957,E2 27954.957} C_VEL
LIN {X 0,Y 620.538,Z 501.987,A -85,B 0,C 180,E1 27952.882,E2 27952.882} C_VEL
LIN {X 0,Y 622.659,Z 358.927,A -85,B 0,C 180,E1 27951.01,E2 27951.01} C_VEL
LIN {X 0,Y 623.157,Z 323.924,A -85,B 0,C 180,E1 27950.511,E2 27950.511} C_VEL
LIN {X 0,Y 622.423,Z 317.936,A -85,B 0,C 180,E1 27950.345,E2 27950.345} C_VEL
LIN {X 0,Y 625.911,Z 290.989,A -85,B 0,C 180,E1 27948.662,E2 27948.662} C_VEL
LIN {X 0,Y 630.454,Z 267.29,A -85,B 0,C 180,E1 27947.033,E2 27947.033} C_VEL
LIN {X 0,Y 628.203,Z 260.386,A -85,B 0,C 180,E1 27945.877,E2 27945.877} C_VEL
LIN {X 0,Y 626.415,Z 255.361,A -85,B 0,C 180,E1 27944.739,E2 27944.739} C_VEL
LIN {X 0,Y 625.348,Z 252.472,A -85,B 0,C 180,E1 27943.816,E2 27943.816} C_VEL
LIN {X 0,Y 624.567,Z 249.826,A -85,B 0,C 180,E1 27942.3,E2 27942.3} C_VEL
LIN {X 0,Y 624.544,Z 249.642,A -85,B 0,C 180,E1 27941.473,E2 27941.473} C_VEL
LIN {X 0,Y 624.752,Z 251.749,A -85,B 0,C 180,E1 27940.091,E2 27940.091} C_VEL
LIN {X 0,Y 625.212,Z 253.057,A -85,B 0,C 180,E1 27939.533,E2 27939.533} C_VEL
LIN {X 0,Y 626.209,Z 256.598,A -85,B 0,C 180,E1 27938.516,E2 27938.516} C_VEL
LIN {X 0,Y 627.862,Z 262.844,A -85,B 0,C 180,E1 27937.241,E2 27937.241} C_VEL
LIN {X 0,Y 628.158,Z 264.412,A -85,B 0,C 180,E1 27936.991,E2 27936.991} C_VEL
LIN {X 0,Y 623.023,Z 289.132,A -85,B 0,C 180,E1 27934.956,E2 27934.956} C_VEL
LIN {X 0,Y 618.197,Z 322.726,A -85,B 0,C 180,E1 27932.403,E2 27932.403} C_VEL
LIN {X 0,Y 614.216,Z 363.397,A -85,B 0,C 180,E1 27929.501,E2 27929.501} C_VEL
LIN {X 0,Y 610.89,Z 409.635,A -85,B 0,C 180,E1 27926.384,E2 27926.384} C_VEL
LIN {X 0,Y 609.712,Z 432.322,A -85,B 0,C 180,E1 27924.921,E2 27924.921} C_VEL
LIN {X 0,Y 613.59,Z 467.49,A -85,B 0,C 180,E1 27923.834,E2 27923.834} C_VEL
LIN {X 0,Y 615.47,Z 490.857,A -85,B 0,C 180,E1 27923.205,E2 27923.205} C_VEL
LIN {X 0,Y 610.773,Z 599.976,A -85,B 0,C 180,E1 27921.289,E2 27921.289} C_VEL
LIN {X 0,Y 608.163,Z 686.24,A -85,B 0,C 180,E1 27919.838,E2 27919.838} C_VEL
LIN {X 0,Y 607.423,Z 708.178,A -85,B 0,C 180,E1 27919.281,E2 27919.281} C_VEL
LIN {X 0,Y 606.694,Z 727.93,A -85,B 0,C 180,E1 27918.602,E2 27918.602} C_VEL
LIN {X 0,Y 605.914,Z 746.818,A -85,B 0,C 180,E1 27917.776,E2 27917.776} C_VEL
LIN {X 0,Y 605.16,Z 764.688,A -85,B 0,C 180,E1 27916.807,E2 27916.807} C_VEL
LIN {X 0,Y 604.392,Z 781.505,A -85,B 0,C 180,E1 27915.693,E2 27915.693} C_VEL
LIN {X 0,Y 603.636,Z 797.159,A -85,B 0,C 180,E1 27914.436,E2 27914.436} C_VEL
LIN {X 0,Y 602.971,Z 810.645,A -85,B 0,C 180,E1 27913.131,E2 27913.131} C_VEL
LIN {X 0,Y 602.351,Z 823.282,A -85,B 0,C 180,E1 27911.653,E2 27911.653} C_VEL
LIN {X 0,Y 601.837,Z 833.841,A -85,B 0,C 180,E1 27910.143,E2 27910.143} C_VEL
LIN {X 0,Y 601.404,Z 843.037,A -85,B 0,C 180,E1 27908.509,E2 27908.509} C_VEL
LIN {X 0,Y 601.1,Z 850.268,A -85,B 0,C 180,E1 27906.879,E2 27906.879} C_VEL
LIN {X 0,Y 600.881,Z 855.972,A -85,B 0,C 180,E1 27905.155,E2 27905.155} C_VEL
LIN {X 0,Y 600.72,Z 859.869,A -85,B 0,C 180,E1 27903.435,E2 27903.435} C_VEL
LIN {X 0,Y 600.611,Z 862.12,A -85,B 0,C 180,E1 27901.622,E2 27901.622} C_VEL
LIN {X 0,Y 600.559,Z 862.545,A -85,B 0,C 180,E1 27899.809,E2 27899.809} C_VEL
LIN {X 0,Y 600.538,Z 861.171,A -85,B 0,C 180,E1 27897.996,E2 27897.996} C_VEL
LIN {X 0,Y 600.564,Z 858.217,A -85,B 0,C 180,E1 27896.277,E2 27896.277} C_VEL
LIN {X 0,Y 600.657,Z 853.536,A -85,B 0,C 180,E1 27894.544,E2 27894.544} C_VEL
LIN {X 0,Y 600.806,Z 847.121,A -85,B 0,C 180,E1 27892.83,E2 27892.83} C_VEL
LIN {X 0,Y 601.056,Z 839.076,A -85,B 0,C 180,E1 27891.172,E2 27891.172} C_VEL
LIN {X 0,Y 601.429,Z 829.289,A -85,B 0,C 180,E1 27889.559,E2 27889.559} C_VEL
LIN {X 0,Y 601.919,Z 817.817,A -85,B 0,C 180,E1 27888.015,E2 27888.015} C_VEL
LIN {X 0,Y 602.52,Z 804.779,A -85,B 0,C 180,E1 27886.566,E2 27886.566} C_VEL
LIN {X 0,Y 603.222,Z 790.109,A -85,B 0,C 180,E1 27885.21,E2 27885.21} C_VEL
LIN {X 0,Y 603.983,Z 774.321,A -85,B 0,C 180,E1 27884,E2 27884} C_VEL
LIN {X 0,Y 604.744,Z 757.506,A -85,B 0,C 180,E1 27882.933,E2 27882.933} C_VEL
LIN {X 0,Y 605.528,Z 739.712,A -85,B 0,C 180,E1 27882.014,E2 27882.014} C_VEL
LIN {X 0,Y 606.282,Z 720.913,A -85,B 0,C 180,E1 27881.24,E2 27881.24} C_VEL
LIN {X 0,Y 606.939,Z 701.311,A -85,B 0,C 180,E1 27880.625,E2 27880.625} C_VEL
LIN {X 0,Y 607.504,Z 680.839,A -85,B 0,C 180,E1 27880.172,E2 27880.172} C_VEL
LIN {X 0,Y 610.916,Z 486.571,A -85,B 0,C 180,E1 27877.445,E2 27877.445} C_VEL
LIN {X 0,Y 607.601,Z 458.258,A -85,B 0,C 180,E1 27876.868,E2 27876.868} C_VEL
LIN {X 0,Y 609.616,Z 407.306,A -85,B 0,C 180,E1 27873.714,E2 27873.714} C_VEL
LIN {X 0,Y 611.998,Z 354.957,A -85,B 0,C 180,E1 27870.435,E2 27870.435} C_VEL
LIN {X 0,Y 613.838,Z 316.525,A -85,B 0,C 180,E1 27867.995,E2 27867.995} C_VEL
LIN {X 0,Y 613.281,Z 310.388,A -85,B 0,C 180,E1 27867.555,E2 27867.555} C_VEL
LIN {X 0,Y 608.553,Z 295.028,A -85,B 0,C 180,E1 27866.249,E2 27866.249} C_VEL
LIN {X 0,Y 608.182,Z 289.748,A -85,B 0,C 180,E1 27865.867,E2 27865.867} C_VEL
LIN {X 0,Y 610.078,Z 254.976,A -85,B 0,C 180,E1 27863.584,E2 27863.584} C_VEL
LIN {X 0,Y 600.345,Z 229.525,A -85,B 0,C 180,E1 27861.136,E2 27861.136} C_VEL
LIN {X 0,Y 593.135,Z 211.351,A -85,B 0,C 180,E1 27859.277,E2 27859.277} C_VEL
LIN {X 0,Y 593.169,Z 211.344,A -85,B 0,C 180,E1 27856.012,E2 27856.012} C_VEL
LIN {X 0,Y 593.18,Z 211.337,A -85,B 0,C 180,E1 27852.84,E2 27852.84} C_VEL
LIN {X 0,Y 593.218,Z 211.467,A -85,B 0,C 180,E1 27851.973,E2 27851.973} C_VEL
LIN {X 0,Y 594.379,Z 214.664,A -85,B 0,C 180,E1 27851.676,E2 27851.676} C_VEL
LIN {X 0,Y 600.487,Z 227.959,A -85,B 0,C 180,E1 27850.303,E2 27850.303} C_VEL
LIN {X 0,Y 607.068,Z 243.692,A -85,B 0,C 180,E1 27848.673,E2 27848.673} C_VEL
LIN {X 0,Y 613.657,Z 261.319,A -85,B 0,C 180,E1 27846.843,E2 27846.843} C_VEL
LIN {X 0,Y 612.425,Z 305.402,A -85,B 0,C 180,E1 27843.662,E2 27843.662} C_VEL
LIN {X 0,Y 612.539,Z 333.426,A -85,B 0,C 180,E1 27841.82,E2 27841.82} C_VEL
LIN {X 0,Y 612.203,Z 336.182,A -85,B 0,C 180,E1 27841.745,E2 27841.745} C_VEL
LIN {X 0,Y 610.183,Z 437.088,A -85,B 0,C 180,E1 27840.402,E2 27840.402} C_VEL
LIN {X 0,Y 607.137,Z 543.148,A -85,B 0,C 180,E1 27838.802,E2 27838.802} C_VEL
LIN {X 0,Y 604.719,Z 624.048,A -85,B 0,C 180,E1 27837.459,E2 27837.459} C_VEL
LIN {X 0,Y 603.991,Z 645.916,A -85,B 0,C 180,E1 27836.926,E2 27836.926} C_VEL
LIN {X 0,Y 603.024,Z 668.157,A -85,B 0,C 180,E1 27836.204,E2 27836.204} C_VEL
LIN {X 0,Y 601.937,Z 689.333,A -85,B 0,C 180,E1 27835.33,E2 27835.33} C_VEL
LIN {X 0,Y 600.766,Z 709.275,A -85,B 0,C 180,E1 27834.326,E2 27834.326} C_VEL
LIN {X 0,Y 599.435,Z 729.797,A -85,B 0,C 180,E1 27833.079,E2 27833.079} C_VEL
LIN {X 0,Y 598.109,Z 749.038,A -85,B 0,C 180,E1 27831.682,E2 27831.682} C_VEL
LIN {X 0,Y 596.935,Z 765.546,A -85,B 0,C 180,E1 27830.277,E2 27830.277} C_VEL
LIN {X 0,Y 595.841,Z 781.606,A -85,B 0,C 180,E1 27828.694,E2 27828.694} C_VEL
LIN {X 0,Y 594.911,Z 795.43,A -85,B 0,C 180,E1 27827.105,E2 27827.105} C_VEL
LIN {X 0,Y 594.069,Z 808.584,A -85,B 0,C 180,E1 27825.322,E2 27825.322} C_VEL
LIN {X 0,Y 593.393,Z 819.658,A -85,B 0,C 180,E1 27823.524,E2 27823.524} C_VEL
LIN {X 0,Y 592.86,Z 829.665,A -85,B 0,C 180,E1 27821.578,E2 27821.578} C_VEL
LIN {X 0,Y 592.523,Z 837.529,A -85,B 0,C 180,E1 27819.715,E2 27819.715} C_VEL
LIN {X 0,Y 592.279,Z 844.168,A -85,B 0,C 180,E1 27817.7,E2 27817.7} C_VEL
LIN {X 0,Y 592.15,Z 849.317,A -85,B 0,C 180,E1 27815.62,E2 27815.62} C_VEL
LIN {X 0,Y 592.102,Z 852.82,A -85,B 0,C 180,E1 27813.582,E2 27813.582} C_VEL
LIN {X 0,Y 592.07,Z 854.699,A -85,B 0,C 180,E1 27811.548,E2 27811.548} C_VEL
LIN {X 0,Y 592.058,Z 855.094,A -85,B 0,C 180,E1 27809.419,E2 27809.419} C_VEL
LIN {X 0,Y 592.081,Z 854.009,A -85,B 0,C 180,E1 27807.387,E2 27807.387} C_VEL
LIN {X 0,Y 592.127,Z 851.322,A -85,B 0,C 180,E1 27805.351,E2 27805.351} C_VEL
LIN {X 0,Y 592.203,Z 846.867,A -85,B 0,C 180,E1 27803.212,E2 27803.212} C_VEL
LIN {X 0,Y 592.383,Z 840.937,A -85,B 0,C 180,E1 27801.164,E2 27801.164} C_VEL
LIN {X 0,Y 592.704,Z 833.557,A -85,B 0,C 180,E1 27799.207,E2 27799.207} C_VEL
LIN {X 0,Y 593.108,Z 824.814,A -85,B 0,C 180,E1 27797.34,E2 27797.34} C_VEL
LIN {X 0,Y 593.707,Z 814.242,A -85,B 0,C 180,E1 27795.467,E2 27795.467} C_VEL
LIN {X 0,Y 594.473,Z 802.239,A -85,B 0,C 180,E1 27793.687,E2 27793.687} C_VEL
LIN {X 0,Y 595.364,Z 788.692,A -85,B 0,C 180,E1 27792,E2 27792} C_VEL
LIN {X 0,Y 596.373,Z 773.725,A -85,B 0,C 180,E1 27790.408,E2 27790.408} C_VEL
LIN {X 0,Y 597.545,Z 756.864,A -85,B 0,C 180,E1 27788.87,E2 27788.87} C_VEL
LIN {X 0,Y 598.763,Z 739.646,A -85,B 0,C 180,E1 27787.517,E2 27787.517} C_VEL
LIN {X 0,Y 600.067,Z 720.184,A -85,B 0,C 180,E1 27786.219,E2 27786.219} C_VEL
LIN {X 0,Y 601.29,Z 700.488,A -85,B 0,C 180,E1 27785.12,E2 27785.12} C_VEL
LIN {X 0,Y 602.434,Z 679.975,A -85,B 0,C 180,E1 27784.171,E2 27784.171} C_VEL
LIN {X 0,Y 603.507,Z 657.848,A -85,B 0,C 180,E1 27783.348,E2 27783.348} C_VEL
LIN {X 0,Y 604.338,Z 636.285,A -85,B 0,C 180,E1 27782.726,E2 27782.726} C_VEL
LIN {X 0,Y 605.009,Z 613.854,A -85,B 0,C 180,E1 27782.258,E2 27782.258} C_VEL
LIN {X 0,Y 608.853,Z 486.088,A -85,B 0,C 180,E1 27780.225,E2 27780.225} C_VEL
LIN {X 0,Y 611.155,Z 394.563,A -85,B 0,C 180,E1 27778.922,E2 27778.922} C_VEL
LIN {X 0,Y 612.283,Z 334.674,A -85,B 0,C 180,E1 27778.137,E2 27778.137} C_VEL
LIN {X 0,Y 612.54,Z 332.282,A -85,B 0,C 180,E1 27778.015,E2 27778.015} C_VEL
LIN {X 0,Y 612.47,Z 304.376,A -85,B 0,C 180,E1 27776.172,E2 27776.172} C_VEL
LIN {X 0,Y 613.671,Z 261.933,A -85,B 0,C 180,E1 27773.106,E2 27773.106} C_VEL
LIN {X 0,Y 612.969,Z 259.122,A -85,B 0,C 180,E1 27772.839,E2 27772.839} C_VEL
LIN {X 0,Y 604.957,Z 238.295,A -85,B 0,C 180,E1 27770.672,E2 27770.672} C_VEL
LIN {X 0,Y 597.566,Z 221.41,A -85,B 0,C 180,E1 27768.922,E2 27768.922} C_VEL
LIN {X 0,Y 594.239,Z 214.4,A -85,B 0,C 180,E1 27768.195,E2 27768.195} C_VEL
LIN {X 0,Y 593.193,Z 211.342,A -85,B 0,C 180,E1 27767.905,E2 27767.905} C_VEL
LIN {X 0,Y 593.178,Z 211.346,A -85,B 0,C 180,E1 27764.656,E2 27764.656} C_VEL
LIN {X 0,Y 593.193,Z 211.34,A -85,B 0,C 180,E1 27761.358,E2 27761.358} C_VEL
LIN {X 0,Y 593.193,Z 211.337,A -85,B 0,C 180,E1 27758.077,E2 27758.077} C_VEL
LIN {X 0,Y 593.177,Z 211.341,A -85,B 0,C 180,E1 27754.824,E2 27754.824} C_VEL
LIN {X 0,Y 593.192,Z 211.337,A -85,B 0,C 180,E1 27751.616,E2 27751.616} C_VEL
LIN {X 0,Y 593.194,Z 211.322,A -85,B 0,C 180,E1 27748.371,E2 27748.371} C_VEL
LIN {X 0,Y 593.186,Z 211.335,A -85,B 0,C 180,E1 27745.03,E2 27745.03} C_VEL
LIN {X 0,Y 593.184,Z 211.337,A -85,B 0,C 180,E1 27741.872,E2 27741.872} C_VEL
LIN {X 0,Y 593.184,Z 211.321,A -85,B 0,C 180,E1 27738.679,E2 27738.679} C_VEL
LIN {X 0,Y 593.185,Z 211.335,A -85,B 0,C 180,E1 27735.446,E2 27735.446} C_VEL
LIN {X 0,Y 593.188,Z 211.315,A -85,B 0,C 180,E1 27732.133,E2 27732.133} C_VEL
LIN {X 0,Y 593.19,Z 211.337,A -85,B 0,C 180,E1 27728.824,E2 27728.824} C_VEL
LIN {X 0,Y 593.172,Z 211.317,A -85,B 0,C 180,E1 27725.708,E2 27725.708} C_VEL
LIN {X 0,Y 593.191,Z 211.34,A -85,B 0,C 180,E1 27722.512,E2 27722.512} C_VEL
LIN {X 0,Y 593.174,Z 211.311,A -85,B 0,C 180,E1 27719.324,E2 27719.324} C_VEL
LIN {X 0,Y 593.186,Z 211.343,A -85,B 0,C 180,E1 27716.037,E2 27716.037} C_VEL
LIN {X 0,Y 593.195,Z 211.309,A -85,B 0,C 180,E1 27712.737,E2 27712.737} C_VEL
LIN {X 0,Y 593.165,Z 211.34,A -85,B 0,C 180,E1 27709.511,E2 27709.511} C_VEL
LIN {X 0,Y 593.199,Z 211.342,A -85,B 0,C 180,E1 27706.251,E2 27706.251} C_VEL
LIN {X 0,Y 593.177,Z 211.339,A -85,B 0,C 180,E1 27703.045,E2 27703.045} C_VEL
LIN {X 0,Y 593.17,Z 211.342,A -85,B 0,C 180,E1 27699.784,E2 27699.784} C_VEL
LIN {X 0,Y 593.201,Z 211.34,A -85,B 0,C 180,E1 27696.559,E2 27696.559} C_VEL
LIN {X 0,Y 593.156,Z 211.336,A -85,B 0,C 180,E1 27693.359,E2 27693.359} C_VEL
LIN {X 0,Y 593.204,Z 211.336,A -85,B 0,C 180,E1 27690.182,E2 27690.182} C_VEL
LIN {X 0,Y 593.162,Z 211.342,A -85,B 0,C 180,E1 27687.011,E2 27687.011} C_VEL
LIN {X 0,Y 593.161,Z 211.34,A -85,B 0,C 180,E1 27683.684,E2 27683.684} C_VEL
LIN {X 0,Y 593.197,Z 211.336,A -85,B 0,C 180,E1 27680.534,E2 27680.534} C_VEL
LIN {X 0,Y 593.157,Z 211.411,A -85,B 0,C 180,E1 27679.366,E2 27679.366} C_VEL
LIN {X 0,Y 594.407,Z 214.747,A -85,B 0,C 180,E1 27679.001,E2 27679.001} C_VEL
LIN {X 0,Y 595.655,Z 216.909,A -85,B 0,C 180,E1 27678.722,E2 27678.722} C_VEL
LIN {X 0,Y 606.616,Z 238.67,A -85,B 0,C 180,E1 27676.188,E2 27676.188} C_VEL
LIN {X 0,Y 617.643,Z 261.089,A -85,B 0,C 180,E1 27673.778,E2 27673.778} C_VEL
LIN {X 0,Y 621.018,Z 268.672,A -85,B 0,C 180,E1 27673.031,E2 27673.031} C_VEL
LIN {X 0,Y 618.145,Z 307.382,A -85,B 0,C 180,E1 27670.934,E2 27670.934} C_VEL
LIN {X 0,Y 620.802,Z 328.6,A -85,B 0,C 180,E1 27670.422,E2 27670.422} C_VEL
LIN {X 0,Y 615.932,Z 572.75,A -85,B 0,C 180,E1 27667.145,E2 27667.145} C_VEL
LIN {X 0,Y 613.838,Z 692.54,A -85,B 0,C 180,E1 27665.574,E2 27665.574} C_VEL
LIN {X 0,Y 612.884,Z 717.171,A -85,B 0,C 180,E1 27665.091,E2 27665.091} C_VEL
LIN {X 0,Y 611.809,Z 738.227,A -85,B 0,C 180,E1 27664.545,E2 27664.545} C_VEL
LIN {X 0,Y 610.287,Z 763.159,A -85,B 0,C 180,E1 27663.724,E2 27663.724} C_VEL
LIN {X 0,Y 608.767,Z 784.121,A -85,B 0,C 180,E1 27662.877,E2 27662.877} C_VEL
LIN {X 0,Y 606.916,Z 808.338,A -85,B 0,C 180,E1 27661.705,E2 27661.705} C_VEL
LIN {X 0,Y 605.256,Z 828.024,A -85,B 0,C 180,E1 27660.585,E2 27660.585} C_VEL
LIN {X 0,Y 603.26,Z 850.119,A -85,B 0,C 180,E1 27659.133,E2 27659.133} C_VEL
LIN {X 0,Y 601.512,Z 869.179,A -85,B 0,C 180,E1 27657.685,E2 27657.685} C_VEL
LIN {X 0,Y 599.633,Z 889.578,A -85,B 0,C 180,E1 27655.905,E2 27655.905} C_VEL
LIN {X 0,Y 598.139,Z 905.898,A -85,B 0,C 180,E1 27654.282,E2 27654.282} C_VEL
LIN {X 0,Y 596.572,Z 923.686,A -85,B 0,C 180,E1 27652.259,E2 27652.259} C_VEL
LIN {X 0,Y 595.456,Z 936.908,A -85,B 0,C 180,E1 27650.546,E2 27650.546} C_VEL
LIN {X 0,Y 594.599,Z 947.776,A -85,B 0,C 180,E1 27648.938,E2 27648.938} C_VEL
LIN {X 0,Y 593.618,Z 960.277,A -85,B 0,C 180,E1 27646.74,E2 27646.74} C_VEL
LIN {X 0,Y 592.984,Z 970.014,A -85,B 0,C 180,E1 27644.751,E2 27644.751} C_VEL
LIN {X 0,Y 592.448,Z 980.189,A -85,B 0,C 180,E1 27642.278,E2 27642.278} C_VEL
LIN {X 0,Y 592.166,Z 987.119,A -85,B 0,C 180,E1 27640.212,E2 27640.212} C_VEL
LIN {X 0,Y 591.983,Z 993.449,A -85,B 0,C 180,E1 27637.863,E2 27637.863} C_VEL
LIN {X 0,Y 591.93,Z 997.654,A -85,B 0,C 180,E1 27635.72,E2 27635.72} C_VEL
LIN {X 0,Y 591.914,Z 1000.463,A -85,B 0,C 180,E1 27633.68,E2 27633.68} C_VEL
LIN {X 0,Y 591.908,Z 1002.213,A -85,B 0,C 180,E1 27631.258,E2 27631.258} C_VEL
LIN {X 0,Y 591.887,Z 1002.326,A -85,B 0,C 180,E1 27629.226,E2 27629.226} C_VEL
LIN {X 0,Y 591.886,Z 1001.29,A -85,B 0,C 180,E1 27627.192,E2 27627.192} C_VEL
LIN {X 0,Y 591.903,Z 998.451,A -85,B 0,C 180,E1 27624.766,E2 27624.766} C_VEL
LIN {X 0,Y 591.965,Z 994.688,A -85,B 0,C 180,E1 27622.722,E2 27622.722} C_VEL
LIN {X 0,Y 592.116,Z 989.184,A -85,B 0,C 180,E1 27620.467,E2 27620.467} C_VEL
LIN {X 0,Y 592.358,Z 981.952,A -85,B 0,C 180,E1 27618.215,E2 27618.215} C_VEL
LIN {X 0,Y 592.718,Z 974.342,A -85,B 0,C 180,E1 27616.24,E2 27616.24} C_VEL
LIN {X 0,Y 593.403,Z 963.252,A -85,B 0,C 180,E1 27613.835,E2 27613.835} C_VEL
LIN {X 0,Y 594.197,Z 952.536,A -85,B 0,C 180,E1 27611.862,E2 27611.862} C_VEL
LIN {X 0,Y 595.198,Z 940.599,A -85,B 0,C 180,E1 27609.958,E2 27609.958} C_VEL
LIN {X 0,Y 596.362,Z 925.486,A -85,B 0,C 180,E1 27608.001,E2 27608.001} C_VEL
LIN {X 0,Y 597.672,Z 909.919,A -85,B 0,C 180,E1 27606.222,E2 27606.222} C_VEL
LIN {X 0,Y 599.159,Z 891.995,A -85,B 0,C 180,E1 27604.444,E2 27604.444} C_VEL
LIN {X 0,Y 600.714,Z 873.905,A -85,B 0,C 180,E1 27602.866,E2 27602.866} C_VEL
LIN {X 0,Y 602.375,Z 853.653,A -85,B 0,C 180,E1 27601.333,E2 27601.333} C_VEL
LIN {X 0,Y 604.021,Z 832.771,A -85,B 0,C 180,E1 27599.955,E2 27599.955} C_VEL
LIN {X 0,Y 605.574,Z 811.745,A -85,B 0,C 180,E1 27598.771,E2 27598.771} C_VEL
LIN {X 0,Y 606.946,Z 791.26,A -85,B 0,C 180,E1 27597.773,E2 27597.773} C_VEL
LIN {X 0,Y 608.392,Z 766.811,A -85,B 0,C 180,E1 27596.777,E2 27596.777} C_VEL
LIN {X 0,Y 609.519,Z 745.309,A -85,B 0,C 180,E1 27596.057,E2 27596.057} C_VEL
LIN {X 0,Y 610.621,Z 720.009,A -85,B 0,C 180,E1 27595.392,E2 27595.392} C_VEL
LIN {X 0,Y 611.316,Z 699.017,A -85,B 0,C 180,E1 27594.976,E2 27594.976} C_VEL
LIN {X 0,Y 611.841,Z 665.599,A -85,B 0,C 180,E1 27594.525,E2 27594.525} C_VEL
LIN {X 0,Y 613.483,Z 505.056,A -85,B 0,C 180,E1 27592.563,E2 27592.563} C_VEL
LIN {X 0,Y 615.769,Z 370.353,A -85,B 0,C 180,E1 27590.755,E2 27590.755} C_VEL
LIN {X 0,Y 616.608,Z 325.242,A -85,B 0,C 180,E1 27590.096,E2 27590.096} C_VEL
LIN {X 0,Y 616.057,Z 320.097,A -85,B 0,C 180,E1 27589.944,E2 27589.944} C_VEL
LIN {X 0,Y 619.827,Z 294.353,A -85,B 0,C 180,E1 27588.284,E2 27588.284} C_VEL
LIN {X 0,Y 624.651,Z 271.49,A -85,B 0,C 180,E1 27586.643,E2 27586.643} C_VEL
LIN {X 0,Y 622.644,Z 264.81,A -85,B 0,C 180,E1 27585.431,E2 27585.431} C_VEL
LIN {X 0,Y 621.136,Z 260.554,A -85,B 0,C 180,E1 27584.319,E2 27584.319} C_VEL
LIN {X 0,Y 620.517,Z 258.704,A -85,B 0,C 180,E1 27583.655,E2 27583.655} C_VEL
LIN {X 0,Y 619.931,Z 256.317,A -85,B 0,C 180,E1 27582.241,E2 27582.241} C_VEL
LIN {X 0,Y 619.921,Z 256.156,A -85,B 0,C 180,E1 27581.523,E2 27581.523} C_VEL
LIN {X 0,Y 620.016,Z 258.169,A -85,B 0,C 180,E1 27580.145,E2 27580.145} C_VEL
LIN {X 0,Y 620.455,Z 259.852,A -85,B 0,C 180,E1 27579.472,E2 27579.472} C_VEL
LIN {X 0,Y 621.477,Z 263.67,A -85,B 0,C 180,E1 27578.392,E2 27578.392} C_VEL
LIN {X 0,Y 622.576,Z 268.976,A -85,B 0,C 180,E1 27577.345,E2 27577.345} C_VEL
LIN {X 0,Y 617.218,Z 291.995,A -85,B 0,C 180,E1 27575.391,E2 27575.391} C_VEL
LIN {X 0,Y 612.142,Z 323.112,A -85,B 0,C 180,E1 27572.952,E2 27572.952} C_VEL
LIN {X 0,Y 607.803,Z 361.756,A -85,B 0,C 180,E1 27570.116,E2 27570.116} C_VEL
LIN {X 0,Y 604.093,Z 407.305,A -85,B 0,C 180,E1 27566.97,E2 27566.97} C_VEL
LIN {X 0,Y 602.826,Z 429.307,A -85,B 0,C 180,E1 27565.521,E2 27565.521} C_VEL
LIN {X 0,Y 606.508,Z 463.394,A -85,B 0,C 180,E1 27564.411,E2 27564.411} C_VEL
LIN {X 0,Y 608.81,Z 491.541,A -85,B 0,C 180,E1 27563.615,E2 27563.615} C_VEL
LIN {X 0,Y 603.933,Z 594.04,A -85,B 0,C 180,E1 27561.749,E2 27561.749} C_VEL
LIN {X 0,Y 600.841,Z 686.375,A -85,B 0,C 180,E1 27560.144,E2 27560.144} C_VEL
LIN {X 0,Y 600.021,Z 708.486,A -85,B 0,C 180,E1 27559.57,E2 27559.57} C_VEL
LIN {X 0,Y 599.252,Z 728.145,A -85,B 0,C 180,E1 27558.887,E2 27558.887} C_VEL
LIN {X 0,Y 598.432,Z 746.855,A -85,B 0,C 180,E1 27558.063,E2 27558.063} C_VEL
LIN {X 0,Y 597.641,Z 764.094,A -85,B 0,C 180,E1 27557.125,E2 27557.125} C_VEL
LIN {X 0,Y 596.819,Z 781.182,A -85,B 0,C 180,E1 27555.998,E2 27555.998} C_VEL
LIN {X 0,Y 596.06,Z 795.961,A -85,B 0,C 180,E1 27554.822,E2 27554.822} C_VEL
LIN {X 0,Y 595.379,Z 808.862,A -85,B 0,C 180,E1 27553.599,E2 27553.599} C_VEL
LIN {X 0,Y 594.741,Z 820.979,A -85,B 0,C 180,E1 27552.23,E2 27552.23} C_VEL
LIN {X 0,Y 594.146,Z 832.402,A -85,B 0,C 180,E1 27550.668,E2 27550.668} C_VEL
LIN {X 0,Y 593.677,Z 841.64,A -85,B 0,C 180,E1 27549.109,E2 27549.109} C_VEL
LIN {X 0,Y 593.308,Z 849.424,A -85,B 0,C 180,E1 27547.456,E2 27547.456} C_VEL
LIN {X 0,Y 593.041,Z 855.653,A -85,B 0,C 180,E1 27545.709,E2 27545.709} C_VEL
LIN {X 0,Y 592.845,Z 860.031,A -85,B 0,C 180,E1 27543.965,E2 27543.965} C_VEL
LIN {X 0,Y 592.713,Z 862.766,A -85,B 0,C 180,E1 27542.127,E2 27542.127} C_VEL
LIN {X 0,Y 592.641,Z 863.646,A -85,B 0,C 180,E1 27540.29,E2 27540.29} C_VEL
LIN {X 0,Y 592.601,Z 862.707,A -85,B 0,C 180,E1 27538.453,E2 27538.453} C_VEL
LIN {X 0,Y 592.619,Z 859.957,A -85,B 0,C 180,E1 27536.614,E2 27536.614} C_VEL
LIN {X 0,Y 592.701,Z 855.339,A -85,B 0,C 180,E1 27534.773,E2 27534.773} C_VEL
LIN {X 0,Y 592.855,Z 849.127,A -85,B 0,C 180,E1 27533.025,E2 27533.025} C_VEL
LIN {X 0,Y 593.118,Z 840.959,A -85,B 0,C 180,E1 27531.273,E2 27531.273} C_VEL
LIN {X 0,Y 593.505,Z 831.215,A -85,B 0,C 180,E1 27529.615,E2 27529.615} C_VEL
LIN {X 0,Y 594.007,Z 819.939,A -85,B 0,C 180,E1 27528.051,E2 27528.051} C_VEL
LIN {X 0,Y 594.621,Z 807.123,A -85,B 0,C 180,E1 27526.582,E2 27526.582} C_VEL
LIN {X 0,Y 595.336,Z 792.725,A -85,B 0,C 180,E1 27525.209,E2 27525.209} C_VEL
LIN {X 0,Y 596.127,Z 777.057,A -85,B 0,C 180,E1 27523.967,E2 27523.967} C_VEL
LIN {X 0,Y 596.94,Z 760.104,A -85,B 0,C 180,E1 27522.854,E2 27522.854} C_VEL
LIN {X 0,Y 597.789,Z 741.744,A -85,B 0,C 180,E1 27521.874,E2 27521.874} C_VEL
LIN {X 0,Y 598.573,Z 723.368,A -85,B 0,C 180,E1 27521.091,E2 27521.091} C_VEL
LIN {X 0,Y 599.278,Z 703.626,A -85,B 0,C 180,E1 27520.443,E2 27520.443} C_VEL
LIN {X 0,Y 599.868,Z 683.691,A -85,B 0,C 180,E1 27519.975,E2 27519.975} C_VEL
LIN {X 0,Y 600.507,Z 648.006,A -85,B 0,C 180,E1 27519.445,E2 27519.445} C_VEL
LIN {X 0,Y 603.646,Z 487.791,A -85,B 0,C 180,E1 27517.152,E2 27517.152} C_VEL
LIN {X 0,Y 600.129,Z 457.216,A -85,B 0,C 180,E1 27516.508,E2 27516.508} C_VEL
LIN {X 0,Y 602.242,Z 407.046,A -85,B 0,C 180,E1 27513.367,E2 27513.367} C_VEL
LIN {X 0,Y 604.811,Z 353.862,A -85,B 0,C 180,E1 27509.999,E2 27509.999} C_VEL
LIN {X 0,Y 607.533,Z 300.915,A -85,B 0,C 180,E1 27506.591,E2 27506.591} C_VEL
LIN {X 0,Y 608.182,Z 289.748,A -85,B 0,C 180,E1 27505.867,E2 27505.867} C_VEL
LIN {X 0,Y 607.662,Z 283.643,A -85,B 0,C 180,E1 27505.418,E2 27505.418} C_VEL
LIN {X 0,Y 603.085,Z 268.41,A -85,B 0,C 180,E1 27504.081,E2 27504.081} C_VEL
LIN {X 0,Y 602.76,Z 263.158,A -85,B 0,C 180,E1 27503.692,E2 27503.692} C_VEL
LIN {X 0,Y 603,Z 258.062,A -85,B 0,C 180,E1 27503.348,E2 27503.348} C_VEL
LIN {X 0,Y 593.193,Z 232.341,A -85,B 0,C 180,E1 27500.84,E2 27500.84} C_VEL
LIN {X 0,Y 585.291,Z 212.68,A -85,B 0,C 180,E1 27498.801,E2 27498.801} C_VEL
LIN {X 0,Y 585.248,Z 212.328,A -85,B 0,C 180,E1 27498.74,E2 27498.74} C_VEL
LIN {X 0,Y 585.242,Z 212.33,A -85,B 0,C 180,E1 27495.534,E2 27495.534} C_VEL
LIN {X 0,Y 585.279,Z 212.511,A -85,B 0,C 180,E1 27492.581,E2 27492.581} C_VEL
LIN {X 0,Y 586.486,Z 215.688,A -85,B 0,C 180,E1 27492.275,E2 27492.275} C_VEL
LIN {X 0,Y 593.915,Z 231.577,A -85,B 0,C 180,E1 27490.598,E2 27490.598} C_VEL
LIN {X 0,Y 600.68,Z 248.052,A -85,B 0,C 180,E1 27488.87,E2 27488.87} C_VEL
LIN {X 0,Y 606.998,Z 264.685,A -85,B 0,C 180,E1 27487.128,E2 27487.128} C_VEL
LIN {X 0,Y 605.845,Z 307.892,A -85,B 0,C 180,E1 27484.021,E2 27484.021} C_VEL
LIN {X 0,Y 605.978,Z 335.125,A -85,B 0,C 180,E1 27482.234,E2 27482.234} C_VEL
LIN {X 0,Y 605.422,Z 338.502,A -85,B 0,C 180,E1 27482.124,E2 27482.124} C_VEL
LIN {X 0,Y 603.338,Z 437.852,A -85,B 0,C 180,E1 27480.788,E2 27480.788} C_VEL
LIN {X 0,Y 600.331,Z 537.417,A -85,B 0,C 180,E1 27479.265,E2 27479.265} C_VEL
LIN {X 0,Y 597.515,Z 624.806,A -85,B 0,C 180,E1 27477.784,E2 27477.784} C_VEL
LIN {X 0,Y 596.746,Z 647.196,A -85,B 0,C 180,E1 27477.232,E2 27477.232} C_VEL
LIN {X 0,Y 595.726,Z 669.58,A -85,B 0,C 180,E1 27476.49,E2 27476.49} C_VEL
LIN {X 0,Y 594.586,Z 690.638,A -85,B 0,C 180,E1 27475.606,E2 27475.606} C_VEL
LIN {X 0,Y 593.358,Z 710.362,A -85,B 0,C 180,E1 27474.597,E2 27474.597} C_VEL
LIN {X 0,Y 592.002,Z 729.982,A -85,B 0,C 180,E1 27473.386,E2 27473.386} C_VEL
LIN {X 0,Y 590.67,Z 747.957,A -85,B 0,C 180,E1 27472.074,E2 27472.074} C_VEL
LIN {X 0,Y 589.337,Z 765.647,A -85,B 0,C 180,E1 27470.561,E2 27470.561} C_VEL
LIN {X 0,Y 588.14,Z 781.742,A -85,B 0,C 180,E1 27468.949,E2 27468.949} C_VEL
LIN {X 0,Y 587.085,Z 796.378,A -85,B 0,C 180,E1 27467.238,E2 27467.238} C_VEL
LIN {X 0,Y 586.208,Z 809.56,A -85,B 0,C 180,E1 27465.432,E2 27465.432} C_VEL
LIN {X 0,Y 585.514,Z 820.562,A -85,B 0,C 180,E1 27463.631,E2 27463.631} C_VEL
LIN {X 0,Y 584.953,Z 830.748,A -85,B 0,C 180,E1 27461.631,E2 27461.631} C_VEL
LIN {X 0,Y 584.605,Z 838.635,A -85,B 0,C 180,E1 27459.749,E2 27459.749} C_VEL
LIN {X 0,Y 584.357,Z 845.109,A -85,B 0,C 180,E1 27457.769,E2 27457.769} C_VEL
LIN {X 0,Y 584.223,Z 850.242,A -85,B 0,C 180,E1 27455.697,E2 27455.697} C_VEL
LIN {X 0,Y 584.169,Z 853.792,A -85,B 0,C 180,E1 27453.631,E2 27453.631} C_VEL
LIN {X 0,Y 584.134,Z 855.693,A -85,B 0,C 180,E1 27451.569,E2 27451.569} C_VEL
LIN {X 0,Y 584.121,Z 856.094,A -85,B 0,C 180,E1 27449.412,E2 27449.412} C_VEL
LIN {X 0,Y 584.145,Z 854.987,A -85,B 0,C 180,E1 27447.351,E2 27447.351} C_VEL
LIN {X 0,Y 584.195,Z 852.266,A -85,B 0,C 180,E1 27445.288,E2 27445.288} C_VEL
LIN {X 0,Y 584.275,Z 847.985,A -85,B 0,C 180,E1 27443.219,E2 27443.219} C_VEL
LIN {X 0,Y 584.455,Z 842.401,A -85,B 0,C 180,E1 27441.242,E2 27441.242} C_VEL
LIN {X 0,Y 584.77,Z 835.046,A -85,B 0,C 180,E1 27439.259,E2 27439.259} C_VEL
LIN {X 0,Y 585.214,Z 825.867,A -85,B 0,C 180,E1 27437.267,E2 27437.267} C_VEL
LIN {X 0,Y 585.834,Z 815.242,A -85,B 0,C 180,E1 27435.368,E2 27435.368} C_VEL
LIN {X 0,Y 586.629,Z 803.187,A -85,B 0,C 180,E1 27433.564,E2 27433.564} C_VEL
LIN {X 0,Y 587.629,Z 788.821,A -85,B 0,C 180,E1 27431.755,E2 27431.755} C_VEL
LIN {X 0,Y 588.721,Z 773.876,A -85,B 0,C 180,E1 27430.143,E2 27430.143} C_VEL
LIN {X 0,Y 589.989,Z 756.998,A -85,B 0,C 180,E1 27428.579,E2 27428.579} C_VEL
LIN {X 0,Y 591.287,Z 739.838,A -85,B 0,C 180,E1 27427.217,E2 27427.217} C_VEL
LIN {X 0,Y 592.627,Z 721.224,A -85,B 0,C 180,E1 27425.954,E2 27425.954} C_VEL
LIN {X 0,Y 593.978,Z 700.668,A -85,B 0,C 180,E1 27424.793,E2 27424.793} C_VEL
LIN {X 0,Y 595.117,Z 681.189,A -85,B 0,C 180,E1 27423.883,E2 27423.883} C_VEL
LIN {X 0,Y 596.2,Z 659.94,A -85,B 0,C 180,E1 27423.075,E2 27423.075} C_VEL
LIN {X 0,Y 597.08,Z 638.557,A -85,B 0,C 180,E1 27422.441,E2 27422.441} C_VEL
LIN {X 0,Y 597.784,Z 616.015,A -85,B 0,C 180,E1 27421.954,E2 27421.954} C_VEL
LIN {X 0,Y 601.653,Z 496.299,A -85,B 0,C 180,E1 27419.995,E2 27419.995} C_VEL
LIN {X 0,Y 604.151,Z 405.264,A -85,B 0,C 180,E1 27418.664,E2 27418.664} C_VEL
LIN {X 0,Y 605.491,Z 337.381,A -85,B 0,C 180,E1 27417.765,E2 27417.765} C_VEL
LIN {X 0,Y 605.977,Z 334.126,A -85,B 0,C 180,E1 27417.61,E2 27417.61} C_VEL
LIN {X 0,Y 605.917,Z 305.223,A -85,B 0,C 180,E1 27415.699,E2 27415.699} C_VEL
LIN {X 0,Y 606.972,Z 264.587,A -85,B 0,C 180,E1 27412.764,E2 27412.764} C_VEL
LIN {X 0,Y 598.693,Z 242.855,A -85,B 0,C 180,E1 27410.482,E2 27410.482} C_VEL
LIN {X 0,Y 590.816,Z 224.56,A -85,B 0,C 180,E1 27408.567,E2 27408.567} C_VEL
LIN {X 0,Y 586.342,Z 215.469,A -85,B 0,C 180,E1 27407.595,E2 27407.595} C_VEL
LIN {X 0,Y 585.243,Z 212.329,A -85,B 0,C 180,E1 27407.279,E2 27407.279} C_VEL
LIN {X 0,Y 585.253,Z 212.321,A -85,B 0,C 180,E1 27404.006,E2 27404.006} C_VEL
LIN {X 0,Y 585.234,Z 212.324,A -85,B 0,C 180,E1 27400.81,E2 27400.81} C_VEL
LIN {X 0,Y 585.255,Z 212.32,A -85,B 0,C 180,E1 27397.559,E2 27397.559} C_VEL
LIN {X 0,Y 585.254,Z 212.324,A -85,B 0,C 180,E1 27394.2,E2 27394.2} C_VEL
LIN {X 0,Y 585.241,Z 212.328,A -85,B 0,C 180,E1 27390.944,E2 27390.944} C_VEL
LIN {X 0,Y 585.247,Z 212.317,A -85,B 0,C 180,E1 27387.692,E2 27387.692} C_VEL
LIN {X 0,Y 585.251,Z 212.313,A -85,B 0,C 180,E1 27384.409,E2 27384.409} C_VEL
LIN {X 0,Y 585.253,Z 212.323,A -85,B 0,C 180,E1 27381.025,E2 27381.025} C_VEL
LIN {X 0,Y 585.241,Z 212.306,A -85,B 0,C 180,E1 27377.808,E2 27377.808} C_VEL
LIN {X 0,Y 585.249,Z 212.328,A -85,B 0,C 180,E1 27374.546,E2 27374.546} C_VEL
LIN {X 0,Y 585.249,Z 212.311,A -85,B 0,C 180,E1 27371.231,E2 27371.231} C_VEL
LIN {X 0,Y 585.244,Z 212.321,A -85,B 0,C 180,E1 27367.955,E2 27367.955} C_VEL
LIN {X 0,Y 585.249,Z 212.31,A -85,B 0,C 180,E1 27364.704,E2 27364.704} C_VEL
LIN {X 0,Y 585.235,Z 212.322,A -85,B 0,C 180,E1 27361.469,E2 27361.469} C_VEL
LIN {X 0,Y 585.253,Z 212.307,A -85,B 0,C 180,E1 27358.238,E2 27358.238} C_VEL
LIN {X 0,Y 585.255,Z 212.323,A -85,B 0,C 180,E1 27354.898,E2 27354.898} C_VEL
LIN {X 0,Y 585.226,Z 212.316,A -85,B 0,C 180,E1 27351.65,E2 27351.65} C_VEL
LIN {X 0,Y 585.257,Z 212.329,A -85,B 0,C 180,E1 27348.469,E2 27348.469} C_VEL
LIN {X 0,Y 585.23,Z 212.325,A -85,B 0,C 180,E1 27345.248,E2 27345.248} C_VEL
LIN {X 0,Y 585.238,Z 212.326,A -85,B 0,C 180,E1 27341.883,E2 27341.883} C_VEL
LIN {X 0,Y 585.261,Z 212.324,A -85,B 0,C 180,E1 27338.66,E2 27338.66} C_VEL
LIN {X 0,Y 585.219,Z 212.33,A -85,B 0,C 180,E1 27335.469,E2 27335.469} C_VEL
LIN {X 0,Y 585.262,Z 212.327,A -85,B 0,C 180,E1 27332.249,E2 27332.249} C_VEL
LIN {X 0,Y 585.224,Z 212.33,A -85,B 0,C 180,E1 27329.051,E2 27329.051} C_VEL
LIN {X 0,Y 585.222,Z 212.33,A -85,B 0,C 180,E1 27325.679,E2 27325.679} C_VEL
LIN {X 0,Y 585.257,Z 212.326,A -85,B 0,C 180,E1 27322.539,E2 27322.539} C_VEL
LIN {X 0,Y 585.261,Z 212.338,A -85,B 0,C 180,E1 27320.094,E2 27320.094} C_VEL
LIN {X 0,Y 586.381,Z 215.581,A -85,B 0,C 180,E1 27319.739,E2 27319.739} C_VEL
LIN {X 0,Y 587.608,Z 217.746,A -85,B 0,C 180,E1 27319.457,E2 27319.457} C_VEL
LIN {X 0,Y 598.082,Z 238.251,A -85,B 0,C 180,E1 27316.991,E2 27316.991} C_VEL
LIN {X 0,Y 610.673,Z 263.873,A -85,B 0,C 180,E1 27314.179,E2 27314.179} C_VEL
LIN {X 0,Y 614.414,Z 272.176,A -85,B 0,C 180,E1 27313.342,E2 27313.342} C_VEL
LIN {X 0,Y 611.616,Z 308.131,A -85,B 0,C 180,E1 27311.376,E2 27311.376} C_VEL
LIN {X 0,Y 614.335,Z 329.922,A -85,B 0,C 180,E1 27310.848,E2 27310.848} C_VEL
LIN {X 0,Y 609.104,Z 573.453,A -85,B 0,C 180,E1 27307.53,E2 27307.53} C_VEL
LIN {X 0,Y 606.877,Z 692.706,A -85,B 0,C 180,E1 27305.945,E2 27305.945} C_VEL
LIN {X 0,Y 605.881,Z 717.138,A -85,B 0,C 180,E1 27305.46,E2 27305.46} C_VEL
LIN {X 0,Y 604.759,Z 738.145,A -85,B 0,C 180,E1 27304.91,E2 27304.91} C_VEL
LIN {X 0,Y 603.156,Z 763.07,A -85,B 0,C 180,E1 27304.078,E2 27304.078} C_VEL
LIN {X 0,Y 601.633,Z 783.135,A -85,B 0,C 180,E1 27303.26,E2 27303.26} C_VEL
LIN {X 0,Y 599.724,Z 806.743,A -85,B 0,C 180,E1 27302.117,E2 27302.117} C_VEL
LIN {X 0,Y 597.919,Z 827.166,A -85,B 0,C 180,E1 27300.946,E2 27300.946} C_VEL
LIN {X 0,Y 595.794,Z 849.632,A -85,B 0,C 180,E1 27299.454,E2 27299.454} C_VEL
LIN {X 0,Y 593.972,Z 868.39,A -85,B 0,C 180,E1 27298.013,E2 27298.013} C_VEL
LIN {X 0,Y 592.002,Z 888.828,A -85,B 0,C 180,E1 27296.211,E2 27296.211} C_VEL
LIN {X 0,Y 590.374,Z 905.637,A -85,B 0,C 180,E1 27294.516,E2 27294.516} C_VEL
LIN {X 0,Y 588.74,Z 923.368,A -85,B 0,C 180,E1 27292.466,E2 27292.466} C_VEL
LIN {X 0,Y 587.493,Z 937.528,A -85,B 0,C 180,E1 27290.596,E2 27290.596} C_VEL
LIN {X 0,Y 586.327,Z 952.004,A -85,B 0,C 180,E1 27288.39,E2 27288.39} C_VEL
LIN {X 0,Y 585.634,Z 961.798,A -85,B 0,C 180,E1 27286.669,E2 27286.669} C_VEL
LIN {X 0,Y 584.963,Z 971.848,A -85,B 0,C 180,E1 27284.553,E2 27284.553} C_VEL
LIN {X 0,Y 584.459,Z 980.895,A -85,B 0,C 180,E1 27282.248,E2 27282.248} C_VEL
LIN {X 0,Y 584.169,Z 987.725,A -85,B 0,C 180,E1 27280.154,E2 27280.154} C_VEL
LIN {X 0,Y 583.971,Z 994.069,A -85,B 0,C 180,E1 27277.675,E2 27277.675} C_VEL
LIN {X 0,Y 583.92,Z 997.973,A -85,B 0,C 180,E1 27275.601,E2 27275.601} C_VEL
LIN {X 0,Y 583.898,Z 1001.016,A -85,B 0,C 180,E1 27273.239,E2 27273.239} C_VEL
LIN {X 0,Y 583.897,Z 1002.28,A -85,B 0,C 180,E1 27270.981,E2 27270.981} C_VEL
LIN {X 0,Y 583.896,Z 1002.28,A -85,B 0,C 180,E1 27269.019,E2 27269.019} C_VEL
LIN {X 0,Y 583.902,Z 1000.914,A -85,B 0,C 180,E1 27266.662,E2 27266.662} C_VEL
LIN {X 0,Y 583.92,Z 997.971,A -85,B 0,C 180,E1 27264.399,E2 27264.399} C_VEL
LIN {X 0,Y 583.972,Z 994.069,A -85,B 0,C 180,E1 27262.325,E2 27262.325} C_VEL
LIN {X 0,Y 584.174,Z 987.581,A -85,B 0,C 180,E1 27259.799,E2 27259.799} C_VEL
LIN {X 0,Y 584.459,Z 980.893,A -85,B 0,C 180,E1 27257.752,E2 27257.752} C_VEL
LIN {X 0,Y 584.963,Z 971.848,A -85,B 0,C 180,E1 27255.447,E2 27255.447} C_VEL
LIN {X 0,Y 585.635,Z 961.803,A -85,B 0,C 180,E1 27253.331,E2 27253.331} C_VEL
LIN {X 0,Y 586.237,Z 953.139,A -85,B 0,C 180,E1 27251.81,E2 27251.81} C_VEL
LIN {X 0,Y 587.284,Z 939.88,A -85,B 0,C 180,E1 27249.78,E2 27249.78} C_VEL
LIN {X 0,Y 588.481,Z 924.956,A -85,B 0,C 180,E1 27247.822,E2 27247.822} C_VEL
LIN {X 0,Y 589.851,Z 909.137,A -85,B 0,C 180,E1 27245.994,E2 27245.994} C_VEL
LIN {X 0,Y 591.407,Z 891.183,A -85,B 0,C 180,E1 27244.192,E2 27244.192} C_VEL
LIN {X 0,Y 593.018,Z 873.034,A -85,B 0,C 180,E1 27242.593,E2 27242.593} C_VEL
LIN {X 0,Y 594.747,Z 852.69,A -85,B 0,C 180,E1 27241.041,E2 27241.041} C_VEL
LIN {X 0,Y 596.345,Z 833.289,A -85,B 0,C 180,E1 27239.745,E2 27239.745} C_VEL
LIN {X 0,Y 598.015,Z 811.764,A -85,B 0,C 180,E1 27238.51,E2 27238.51} C_VEL
LIN {X 0,Y 599.428,Z 791.633,A -85,B 0,C 180,E1 27237.512,E2 27237.512} C_VEL
LIN {X 0,Y 601.005,Z 766.513,A -85,B 0,C 180,E1 27236.472,E2 27236.472} C_VEL
LIN {X 0,Y 602.239,Z 744.264,A -85,B 0,C 180,E1 27235.718,E2 27235.718} C_VEL
LIN {X 0,Y 603.361,Z 719.506,A -85,B 0,C 180,E1 27235.064,E2 27235.064} C_VEL
LIN {X 0,Y 604.09,Z 698.59,A -85,B 0,C 180,E1 27234.645,E2 27234.645} C_VEL
LIN {X 0,Y 604.653,Z 664.91,A -85,B 0,C 180,E1 27234.185,E2 27234.185} C_VEL
LIN {X 0,Y 606.419,Z 513.799,A -85,B 0,C 180,E1 27232.303,E2 27232.303} C_VEL
LIN {X 0,Y 608.891,Z 383.836,A -85,B 0,C 180,E1 27230.519,E2 27230.519} C_VEL
LIN {X 0,Y 610.213,Z 326.648,A -85,B 0,C 180,E1 27229.66,E2 27229.66} C_VEL
LIN {X 0,Y 609.782,Z 322.554,A -85,B 0,C 180,E1 27229.539,E2 27229.539} C_VEL
LIN {X 0,Y 613.985,Z 297.393,A -85,B 0,C 180,E1 27227.859,E2 27227.859} C_VEL
LIN {X 0,Y 619.057,Z 276.157,A -85,B 0,C 180,E1 27226.299,E2 27226.299} C_VEL
LIN {X 0,Y 617.446,Z 270.406,A -85,B 0,C 180,E1 27225.178,E2 27225.178} C_VEL
LIN {X 0,Y 616.157,Z 266.128,A -85,B 0,C 180,E1 27223.992,E2 27223.992} C_VEL
LIN {X 0,Y 615.288,Z 263.382,A -85,B 0,C 180,E1 27222.595,E2 27222.595} C_VEL
LIN {X 0,Y 615.355,Z 262.551,A -85,B 0,C 180,E1 27221.769,E2 27221.769} C_VEL
LIN {X 0,Y 615.239,Z 264.441,A -85,B 0,C 180,E1 27220.303,E2 27220.303} C_VEL
LIN {X 0,Y 615.563,Z 265.9,A -85,B 0,C 180,E1 27219.651,E2 27219.651} C_VEL
LIN {X 0,Y 616.38,Z 269.551,A -85,B 0,C 180,E1 27218.565,E2 27218.565} C_VEL
LIN {X 0,Y 617.125,Z 273.642,A -85,B 0,C 180,E1 27217.708,E2 27217.708} C_VEL
LIN {X 0,Y 611.54,Z 295.137,A -85,B 0,C 180,E1 27215.827,E2 27215.827} C_VEL
LIN {X 0,Y 606.196,Z 324.086,A -85,B 0,C 180,E1 27213.487,E2 27213.487} C_VEL
LIN {X 0,Y 601.464,Z 361.147,A -85,B 0,C 180,E1 27210.688,E2 27210.688} C_VEL
LIN {X 0,Y 597.304,Z 406.578,A -85,B 0,C 180,E1 27207.473,E2 27207.473} C_VEL
LIN {X 0,Y 596.036,Z 426.295,A -85,B 0,C 180,E1 27206.149,E2 27206.149} C_VEL
LIN {X 0,Y 599.748,Z 461.707,A -85,B 0,C 180,E1 27204.939,E2 27204.939} C_VEL
LIN {X 0,Y 602.193,Z 492.466,A -85,B 0,C 180,E1 27204.033,E2 27204.033} C_VEL
LIN {X 0,Y 596.686,Z 600.228,A -85,B 0,C 180,E1 27202.011,E2 27202.011} C_VEL
LIN {X 0,Y 593.541,Z 686.878,A -85,B 0,C 180,E1 27200.454,E2 27200.454} C_VEL
LIN {X 0,Y 592.663,Z 709.153,A -85,B 0,C 180,E1 27199.865,E2 27199.865} C_VEL
LIN {X 0,Y 591.792,Z 729.638,A -85,B 0,C 180,E1 27199.134,E2 27199.134} C_VEL
LIN {X 0,Y 590.868,Z 749.261,A -85,B 0,C 180,E1 27198.244,E2 27198.244} C_VEL
LIN {X 0,Y 590.016,Z 766.959,A -85,B 0,C 180,E1 27197.252,E2 27197.252} C_VEL
LIN {X 0,Y 589.169,Z 783.254,A -85,B 0,C 180,E1 27196.143,E2 27196.143} C_VEL
LIN {X 0,Y 588.317,Z 798.784,A -85,B 0,C 180,E1 27194.871,E2 27194.871} C_VEL
LIN {X 0,Y 587.535,Z 812.852,A -85,B 0,C 180,E1 27193.483,E2 27193.483} C_VEL
LIN {X 0,Y 586.836,Z 825.27,A -85,B 0,C 180,E1 27191.998,E2 27191.998} C_VEL
LIN {X 0,Y 586.228,Z 836.085,A -85,B 0,C 180,E1 27190.416,E2 27190.416} C_VEL
LIN {X 0,Y 585.724,Z 845.362,A -85,B 0,C 180,E1 27188.73,E2 27188.73} C_VEL
LIN {X 0,Y 585.36,Z 852.612,A -85,B 0,C 180,E1 27187.047,E2 27187.047} C_VEL
LIN {X 0,Y 585.097,Z 858.237,A -85,B 0,C 180,E1 27185.295,E2 27185.295} C_VEL
LIN {X 0,Y 584.899,Z 862.098,A -85,B 0,C 180,E1 27183.528,E2 27183.528} C_VEL
LIN {X 0,Y 584.764,Z 864.292,A -85,B 0,C 180,E1 27181.666,E2 27181.666} C_VEL
LIN {X 0,Y 584.702,Z 864.684,A -85,B 0,C 180,E1 27179.902,E2 27179.902} C_VEL
LIN {X 0,Y 584.671,Z 863.3,A -85,B 0,C 180,E1 27178.04,E2 27178.04} C_VEL
LIN {X 0,Y 584.698,Z 860.087,A -85,B 0,C 180,E1 27176.176,E2 27176.176} C_VEL
LIN {X 0,Y 584.801,Z 855.3,A -85,B 0,C 180,E1 27174.407,E2 27174.407} C_VEL
LIN {X 0,Y 584.974,Z 848.69,A -85,B 0,C 180,E1 27172.635,E2 27172.635} C_VEL
LIN {X 0,Y 585.275,Z 840.066,A -85,B 0,C 180,E1 27170.858,E2 27170.858} C_VEL
LIN {X 0,Y 585.712,Z 829.836,A -85,B 0,C 180,E1 27169.176,E2 27169.176} C_VEL
LIN {X 0,Y 586.274,Z 818.03,A -85,B 0,C 180,E1 27167.591,E2 27167.591} C_VEL
LIN {X 0,Y 586.985,Z 804.127,A -85,B 0,C 180,E1 27166.052,E2 27166.052} C_VEL
LIN {X 0,Y 587.785,Z 789.01,A -85,B 0,C 180,E1 27164.666,E2 27164.666} C_VEL
LIN {X 0,Y 588.613,Z 773.301,A -85,B 0,C 180,E1 27163.469,E2 27163.469} C_VEL
LIN {X 0,Y 589.473,Z 755.981,A -85,B 0,C 180,E1 27162.375,E2 27162.375} C_VEL
LIN {X 0,Y 590.364,Z 737.587,A -85,B 0,C 180,E1 27161.433,E2 27161.433} C_VEL
LIN {X 0,Y 591.164,Z 718.702,A -85,B 0,C 180,E1 27160.667,E2 27160.667} C_VEL
LIN {X 0,Y 591.869,Z 698.765,A -85,B 0,C 180,E1 27160.056,E2 27160.056} C_VEL
LIN {X 0,Y 592.457,Z 678.561,A -85,B 0,C 180,E1 27159.623,E2 27159.623} C_VEL
LIN {X 0,Y 596.329,Z 488.725,A -85,B 0,C 180,E1 27156.851,E2 27156.851} C_VEL
LIN {X 0,Y 592.66,Z 456.622,A -85,B 0,C 180,E1 27156.167,E2 27156.167} C_VEL
LIN {X 0,Y 594.885,Z 406.758,A -85,B 0,C 180,E1 27153.011,E2 27153.011} C_VEL
LIN {X 0,Y 597.647,Z 352.544,A -85,B 0,C 180,E1 27149.54,E2 27149.54} C_VEL
LIN {X 0,Y 600.505,Z 300.475,A -85,B 0,C 180,E1 27146.153,E2 27146.153} C_VEL
LIN {X 0,Y 602.76,Z 263.158,A -85,B 0,C 180,E1 27143.692,E2 27143.692} C_VEL
LIN {X 0,Y 602.249,Z 260.454,A -85,B 0,C 180,E1 27143.469,E2 27143.469} C_VEL
LIN {X 0,Y 599.563,Z 257.226,A -85,B 0,C 180,E1 27143.067,E2 27143.067} C_VEL
LIN {X 0,Y 593.361,Z 252.549,A -85,B 0,C 180,E1 27142.324,E2 27142.324} C_VEL
LIN {X 0,Y 591.877,Z 250.242,A -85,B 0,C 180,E1 27142.056,E2 27142.056} C_VEL
LIN {X 0,Y 582.778,Z 227.034,A -85,B 0,C 180,E1 27139.697,E2 27139.697} C_VEL
LIN {X 0,Y 577.284,Z 213.321,A -85,B 0,C 180,E1 27138.209,E2 27138.209} C_VEL
LIN {X 0,Y 577.318,Z 213.312,A -85,B 0,C 180,E1 27135.038,E2 27135.038} C_VEL
LIN {X 0,Y 577.306,Z 213.326,A -85,B 0,C 180,E1 27133.23,E2 27133.23} C_VEL
LIN {X 0,Y 578.39,Z 216.458,A -85,B 0,C 180,E1 27132.932,E2 27132.932} C_VEL
LIN {X 0,Y 579.741,Z 219.06,A -85,B 0,C 180,E1 27132.642,E2 27132.642} C_VEL
LIN {X 0,Y 587.775,Z 236.28,A -85,B 0,C 180,E1 27130.798,E2 27130.798} C_VEL
LIN {X 0,Y 595.769,Z 256.018,A -85,B 0,C 180,E1 27128.701,E2 27128.701} C_VEL
LIN {X 0,Y 600.354,Z 268.408,A -85,B 0,C 180,E1 27127.397,E2 27127.397} C_VEL
LIN {X 0,Y 599.285,Z 311.246,A -85,B 0,C 180,E1 27124.329,E2 27124.329} C_VEL
LIN {X 0,Y 599.439,Z 336.798,A -85,B 0,C 180,E1 27122.657,E2 27122.657} C_VEL
LIN {X 0,Y 598.667,Z 341.014,A -85,B 0,C 180,E1 27122.508,E2 27122.508} C_VEL
LIN {X 0,Y 596.521,Z 438.755,A -85,B 0,C 180,E1 27121.181,E2 27121.181} C_VEL
LIN {X 0,Y 593.543,Z 532.789,A -85,B 0,C 180,E1 27119.723,E2 27119.723} C_VEL
LIN {X 0,Y 590.364,Z 624.995,A -85,B 0,C 180,E1 27118.131,E2 27118.131} C_VEL
LIN {X 0,Y 589.56,Z 647.957,A -85,B 0,C 180,E1 27117.563,E2 27117.563} C_VEL
LIN {X 0,Y 588.536,Z 669.721,A -85,B 0,C 180,E1 27116.84,E2 27116.84} C_VEL
LIN {X 0,Y 587.392,Z 690.277,A -85,B 0,C 180,E1 27115.977,E2 27115.977} C_VEL
LIN {X 0,Y 586.04,Z 710.662,A -85,B 0,C 180,E1 27114.925,E2 27114.925} C_VEL
LIN {X 0,Y 584.669,Z 729.58,A -85,B 0,C 180,E1 27113.75,E2 27113.75} C_VEL
LIN {X 0,Y 583.248,Z 747.753,A -85,B 0,C 180,E1 27112.423,E2 27112.423} C_VEL
LIN {X 0,Y 581.878,Z 765.048,A -85,B 0,C 180,E1 27110.942,E2 27110.942} C_VEL
LIN {X 0,Y 580.654,Z 780.427,A -85,B 0,C 180,E1 27109.411,E2 27109.411} C_VEL
LIN {X 0,Y 579.482,Z 795.245,A -85,B 0,C 180,E1 27107.679,E2 27107.679} C_VEL
LIN {X 0,Y 578.55,Z 807.897,A -85,B 0,C 180,E1 27105.95,E2 27105.95} C_VEL
LIN {X 0,Y 577.748,Z 819.913,A -85,B 0,C 180,E1 27104.022,E2 27104.022} C_VEL
LIN {X 0,Y 577.166,Z 829.985,A -85,B 0,C 180,E1 27102.1,E2 27102.1} C_VEL
LIN {X 0,Y 576.749,Z 838.161,A -85,B 0,C 180,E1 27100.185,E2 27100.185} C_VEL
LIN {X 0,Y 576.472,Z 845.031,A -85,B 0,C 180,E1 27098.177,E2 27098.177} C_VEL
LIN {X 0,Y 576.332,Z 850.343,A -85,B 0,C 180,E1 27096.175,E2 27096.175} C_VEL
LIN {X 0,Y 576.238,Z 854.154,A -85,B 0,C 180,E1 27094.08,E2 27094.08} C_VEL
LIN {X 0,Y 576.207,Z 856.482,A -85,B 0,C 180,E1 27091.889,E2 27091.889} C_VEL
LIN {X 0,Y 576.199,Z 857.182,A -85,B 0,C 180,E1 27089.801,E2 27089.801} C_VEL
LIN {X 0,Y 576.204,Z 856.281,A -85,B 0,C 180,E1 27087.713,E2 27087.713} C_VEL
LIN {X 0,Y 576.248,Z 853.833,A -85,B 0,C 180,E1 27085.621,E2 27085.621} C_VEL
LIN {X 0,Y 576.344,Z 849.843,A -85,B 0,C 180,E1 27083.525,E2 27083.525} C_VEL
LIN {X 0,Y 576.515,Z 844.122,A -85,B 0,C 180,E1 27081.422,E2 27081.422} C_VEL
LIN {X 0,Y 576.818,Z 836.801,A -85,B 0,C 180,E1 27079.382,E2 27079.382} C_VEL
LIN {X 0,Y 577.289,Z 827.415,A -85,B 0,C 180,E1 27077.293,E2 27077.293} C_VEL
LIN {X 0,Y 577.934,Z 816.921,A -85,B 0,C 180,E1 27075.369,E2 27075.369} C_VEL
LIN {X 0,Y 578.818,Z 804.354,A -85,B 0,C 180,E1 27073.439,E2 27073.439} C_VEL
LIN {X 0,Y 579.816,Z 790.982,A -85,B 0,C 180,E1 27071.708,E2 27071.708} C_VEL
LIN {X 0,Y 580.962,Z 776.343,A -85,B 0,C 180,E1 27070.076,E2 27070.076} C_VEL
LIN {X 0,Y 582.298,Z 759.809,A -85,B 0,C 180,E1 27068.493,E2 27068.493} C_VEL
LIN {X 0,Y 583.711,Z 742.222,A -85,B 0,C 180,E1 27067.054,E2 27067.054} C_VEL
LIN {X 0,Y 585.156,Z 723.193,A -85,B 0,C 180,E1 27065.735,E2 27065.735} C_VEL
LIN {X 0,Y 586.509,Z 703.816,A -85,B 0,C 180,E1 27064.611,E2 27064.611} C_VEL
LIN {X 0,Y 587.764,Z 683.712,A -85,B 0,C 180,E1 27063.64,E2 27063.64} C_VEL
LIN {X 0,Y 588.932,Z 661.915,A -85,B 0,C 180,E1 27062.789,E2 27062.789} C_VEL
LIN {X 0,Y 589.873,Z 640.331,A -85,B 0,C 180,E1 27062.133,E2 27062.133} C_VEL
LIN {X 0,Y 590.601,Z 617.84,A -85,B 0,C 180,E1 27061.635,E2 27061.635} C_VEL
LIN {X 0,Y 594.551,Z 503.519,A -85,B 0,C 180,E1 27059.714,E2 27059.714} C_VEL
LIN {X 0,Y 597.181,Z 414.489,A -85,B 0,C 180,E1 27058.382,E2 27058.382} C_VEL
LIN {X 0,Y 598.837,Z 339.586,A -85,B 0,C 180,E1 27057.363,E2 27057.363} C_VEL
LIN {X 0,Y 599.448,Z 336.228,A -85,B 0,C 180,E1 27057.213,E2 27057.213} C_VEL
LIN {X 0,Y 599.375,Z 306.855,A -85,B 0,C 180,E1 27055.271,E2 27055.271} C_VEL
LIN {X 0,Y 600.383,Z 268.326,A -85,B 0,C 180,E1 27052.498,E2 27052.498} C_VEL
